KUKA KRL program: MyProgram_092().src

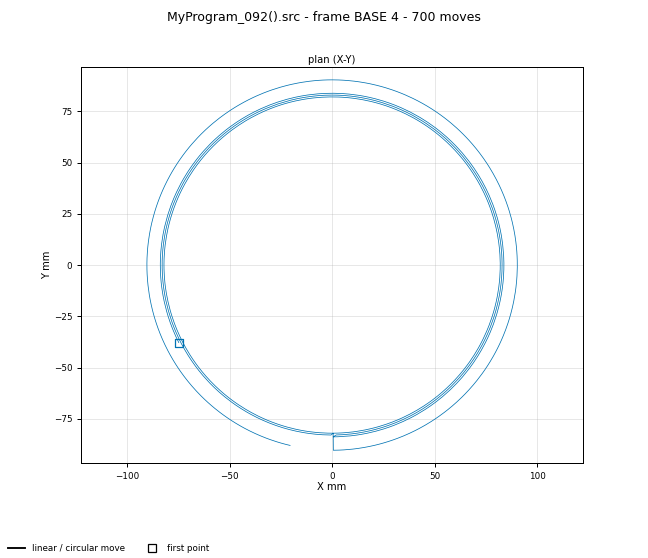
[picture p0: tool path of MyProgram_092().src in frame BASE 4, 700 of 700 moves have a stored position in this frame; points joined in program order, loops and branches not executed]
&ACCESS RVP
&REL 1
&PARAM TEMPLATE = C:\KRC\Roboter\Template\vorgabe
&PARAM EDITMASK = *
DEF MyProgram_092()
; ---- Setting reference (Base) ----
$BASE = BASE_DATA[4]

; --------------------------
; ---- Setting tool (TCP) ----
$TOOL = TOOL_DATA[3]
; --------------------------

$VEL.CP = VEL_APROX_PRINT
Startdeposition()
$VEL.CP = VEL_PRINT
LIN {X -74.828,Y -37.8282,Z 87,A -158.7584,B 24.9189,C -2.0802,E1 24.8563,E2 243.6594} C_DIS
LIN {X -76.2325,Y -34.9131,Z 87,A -161.0575,B 24.9186,C -2.084,E1 24.8536,E2 245.962} C_DIS
LIN {X -77.7703,Y -31.3357,Z 87,A -163.8809,B 24.9183,C -2.0873,E1 24.8506,E2 248.7932} C_DIS
LIN {X -78.9715,Y -28.1737,Z 87,A -166.4538,B 24.9183,C -2.0871,E1 24.8481,E2 251.3812} C_DIS
LIN {X -80.015,Y -25.0533,Z 87,A -168.1806,B 24.9167,C -2.1077,E1 24.8467,E2 253.0687} C_DIS
LIN {X -80.7299,Y -22.6451,Z 87,A -169.9657,B 24.9164,C -2.111,E1 24.8453,E2 254.8562} C_DIS
LIN {X -81.9682,Y -17.6447,Z 87,A -173.2787,B 24.9151,C -2.1273,E1 24.8432,E2 258.1497} C_DIS
LIN {X -82.5461,Y -14.7049,Z 87,A -175.5042,B 24.9151,C -2.1289,E1 24.842,E2 260.3846} C_DIS
LIN {X -83.1122,Y -11.0688,Z 87,A -177.8414,B 24.914,C -2.1414,E1 24.8411,E2 262.7057} C_DIS
LIN {X -83.3919,Y -8.7092,Z 87,A -179.5472,B 24.9138,C -2.1444,E1 24.8405,E2 264.4148} C_DIS
LIN {X -83.6299,Y -6.0204,Z 87,A 178.4494,B 24.9136,C -2.146,E1 24.8401,E2 266.4264} C_DIS
LIN {X -83.7977,Y -2.8427,Z 87,A 176.1823,B 24.9133,C -2.1504,E1 24.8398,E2 268.6965} C_DIS
LIN {X -83.8443,Y 0.5678,Z 87,A 174.0248,B 24.9123,C -2.1624,E1 24.8398,E2 270.8383} C_DIS
LIN {X -83.7774,Y 3.3843,Z 87,A 172.0675,B 24.9119,C -2.1678,E1 24.84,E2 272.7947} C_DIS
LIN {X -83.5899,Y 6.5428,Z 87,A 169.334,B 24.9125,C -2.1596,E1 24.8405,E2 275.5641} C_DIS
LIN {X -83.2161,Y 10.2664,Z 87,A 166.7868,B 24.9118,C -2.168,E1 24.8414,E2 278.1066} C_DIS
LIN {X -82.5012,Y 14.9543,Z 87,A 163.3356,B 24.9114,C -2.1728,E1 24.843,E2 281.5668} C_DIS
LIN {X -81.7692,Y 18.5465,Z 87,A 161.7678,B 24.9088,C -2.2054,E1 24.8439,E2 283.0659} C_DIS
LIN {X -80.2055,Y 24.4398,Z 87,A 157.3428,B 24.9083,C -2.2116,E1 24.8472,E2 287.5019} C_DIS
LIN {X -78.6612,Y 29.0272,Z 87,A 154.246,B 24.9069,C -2.2274,E1 24.8499,E2 290.5785} C_DIS
LIN {X -77.2818,Y 32.5206,Z 87,A 151.4219,B 24.9069,C -2.2283,E1 24.8529,E2 293.4163} C_DIS
LIN {X -75.9355,Y 35.5514,Z 87,A 148.0998,B 24.9086,C -2.2072,E1 24.8569,E2 296.8069} C_DIS
LIN {X -73.8493,Y 39.7045,Z 87,A 146.1931,B 24.905,C -2.2501,E1 24.8592,E2 298.6214} C_DIS
LIN {X -72.4886,Y 42.1385,Z 87,A 144.1984,B 24.9048,C -2.2531,E1 24.862,E2 300.6192} C_DIS
LIN {X -70.5351,Y 45.3307,Z 87,A 141.4848,B 24.9045,C -2.2562,E1 24.866,E2 303.3394} C_DIS
LIN {X -68.5387,Y 48.2985,Z 87,A 138.87,B 24.9043,C -2.2583,E1 24.8701,E2 305.9622} C_DIS
LIN {X -66.2293,Y 51.4182,Z 87,A 136.4276,B 24.9032,C -2.271,E1 24.8742,E2 308.3859} C_DIS
LIN {X -64.7484,Y 53.2718,Z 87,A 134.6169,B 24.9033,C -2.2701,E1 24.8774,E2 310.2071} C_DIS
LIN {X -62.7537,Y 55.6077,Z 87,A 132.2198,B 24.9036,C -2.2674,E1 24.8818,E2 312.6217} C_DIS
LIN {X -59.4872,Y 59.088,Z 87,A 129.4081,B 24.9018,C -2.2875,E1 24.8872,E2 315.3974} C_DIS
LIN {X -57.6192,Y 60.911,Z 87,A 127.4312,B 24.9019,C -2.2865,E1 24.8912,E2 317.385} C_DIS
LIN {X -55.0222,Y 63.2665,Z 87,A 124.7933,B 24.902,C -2.2853,E1 24.8967,E2 320.0362} C_DIS
LIN {X -51.7994,Y 65.9314,Z 87,A 122.4481,B 24.9003,C -2.3055,E1 24.9017,E2 322.342} C_DIS
LIN {X -49.9627,Y 67.3352,Z 87,A 120.4367,B 24.901,C -2.2969,E1 24.9063,E2 324.3812} C_DIS
LIN {X -46.6431,Y 69.6755,Z 87,A 117.8495,B 24.9001,C -2.3076,E1 24.9122,E2 326.9517} C_DIS
LIN {X -43.9616,Y 71.3981,Z 87,A 115.5051,B 24.9001,C -2.307,E1 24.9178,E2 329.3048} C_DIS
LIN {X -40.9981,Y 73.1385,Z 87,A 112.6787,B 24.9009,C -2.2979,E1 24.9247,E2 332.1612} C_DIS
LIN {X -38.0284,Y 74.7257,Z 87,A 111.0801,B 24.8989,C -2.3212,E1 24.9285,E2 333.7087} C_DIS
LIN {X -34.9535,Y 76.2138,Z 87,A 108.7935,B 24.8985,C -2.3261,E1 24.9343,E2 335.9894} C_DIS
LIN {X -30.3308,Y 78.1669,Z 87,A 104.6708,B 24.8998,C -2.3114,E1 24.945,E2 340.1564} C_DIS
LIN {X -26.6364,Y 79.5022,Z 87,A 101.4349,B 24.9008,C -2.2992,E1 24.9537,E2 343.4274} C_DIS
LIN {X -22.04,Y 80.8971,Z 87,A 99.0674,B 24.8983,C -2.3285,E1 24.9599,E2 345.729} C_DIS
LIN {X -18.0377,Y 81.8825,Z 87,A 96.3469,B 24.8978,C -2.3338,E1 24.9673,E2 348.4404} C_DIS
LIN {X -15.0523,Y 82.4836,Z 87,A 94.3269,B 24.8975,C -2.3372,E1 24.9728,E2 350.4545} C_DIS
LIN {X -11.9026,Y 82.9964,Z 87,A 91.9253,B 24.8979,C -2.3323,E1 24.9794,E2 352.8699} C_DIS
LIN {X -7.092,Y 83.546,Z 87,A 89.013,B 24.8968,C -2.3456,E1 24.9875,E2 355.7524} C_DIS
LIN {X -3.5283,Y 83.7712,Z 87,A 86.3333,B 24.8973,C -2.3395,E1 24.995,E2 358.4473} C_DIS
LIN {X 0.6383,Y 83.8431,Z 87,A 82.993,B 24.8985,C -2.3256,E1 25.0044,E2 361.8205} C_DIS
LIN {X 4.9069,Y 83.7022,Z 87,A 80.4957,B 24.8974,C -2.3382,E1 25.0113,E2 364.2872} C_DIS
LIN {X 8.2541,Y 83.4395,Z 87,A 77.7923,B 24.8985,C -2.3258,E1 25.0189,E2 367.0184} C_DIS
LIN {X 13.1274,Y 82.8121,Z 87,A 74.8322,B 24.8975,C -2.3368,E1 25.027,E2 369.9498} C_DIS
LIN {X 15.5161,Y 82.398,Z 87,A 73.2663,B 24.8974,C -2.3389,E1 25.0312,E2 371.509} C_DIS
LIN {X 18.3808,Y 81.8075,Z 87,A 71.2516,B 24.8974,C -2.3374,E1 25.0367,E2 373.5245} C_DIS
LIN {X 21.1726,Y 81.1288,Z 87,A 68.9963,B 24.8984,C -2.3274,E1 25.0429,E2 375.8001} C_DIS
LIN {X 24.9022,Y 80.0622,Z 87,A 66.3151,B 24.8986,C -2.3246,E1 25.0501,E2 378.4834} C_DIS
LIN {X 28.008,Y 79.0296,Z 87,A 64.3946,B 24.8979,C -2.3323,E1 25.0551,E2 380.3818} C_DIS
LIN {X 30.6424,Y 78.0456,Z 87,A 62.5561,B 24.8979,C -2.333,E1 25.0599,E2 382.2146} C_DIS
LIN {X 33.5893,Y 76.8234,Z 87,A 60.3428,B 24.8982,C -2.3296,E1 25.0656,E2 384.4305} C_DIS
LIN {X 37.9144,Y 74.784,Z 87,A 57.3959,B 24.8976,C -2.3357,E1 25.0729,E2 387.3554} C_DIS
LIN {X 42.9467,Y 72.0122,Z 87,A 52.651,B 24.9003,C -2.3047,E1 25.0846,E2 392.1597} C_DIS
LIN {X 46.689,Y 69.6444,Z 87,A 49.1059,B 24.9022,C -2.2837,E1 25.0929,E2 395.7426} C_DIS
LIN {X 50.6024,Y 66.8547,Z 87,A 47.0392,B 24.8993,C -2.3162,E1 25.0974,E2 397.7252} C_DIS
LIN {X 52.6102,Y 65.2862,Z 87,A 45.1077,B 24.9001,C -2.3069,E1 25.1016,E2 399.6713} C_DIS
LIN {X 55.6902,Y 62.6799,Z 87,A 42.3443,B 24.9006,C -2.3014,E1 25.1075,E2 402.437} C_DIS
LIN {X 58.1521,Y 60.402,Z 87,A 40.1346,B 24.9008,C -2.2994,E1 25.112,E2 404.6424} C_DIS
LIN {X 60.4415,Y 58.1111,Z 87,A 37.9335,B 24.9012,C -2.295,E1 25.1163,E2 406.8444} C_DIS
LIN {X 63.4897,Y 54.7666,Z 87,A 34.9971,B 24.9013,C -2.2931,E1 25.1217,E2 409.7722} C_DIS
LIN {X 66.8785,Y 50.5707,Z 87,A 30.8014,B 24.9035,C -2.2679,E1 25.1291,E2 414.0078} C_DIS
LIN {X 69.2571,Y 47.2612,Z 87,A 27.9992,B 24.9042,C -2.2603,E1 25.1335,E2 416.8142} C_DIS
LIN {X 71.484,Y 43.8202,Z 87,A 25.6091,B 24.9036,C -2.2664,E1 25.1371,E2 419.1779} C_DIS
LIN {X 73.1323,Y 41.0092,Z 87,A 22.6384,B 24.9062,C -2.2363,E1 25.1412,E2 422.2042} C_DIS
LIN {X 74.9856,Y 37.5142,Z 87,A 21.0042,B 24.9039,C -2.2637,E1 25.1432,E2 423.765} C_DIS
LIN {X 76.5866,Y 34.1275,Z 87,A 17.8198,B 24.9062,C -2.236,E1 25.147,E2 426.9976} C_DIS
LIN {X 78.3944,Y 29.7386,Z 87,A 15.0097,B 24.9058,C -2.2409,E1 25.1499,E2 429.7806} C_DIS
LIN {X 79.4552,Y 26.7757,Z 87,A 12.8323,B 24.9064,C -2.2337,E1 25.1519,E2 431.9629} C_DIS
LIN {X 80.6296,Y 22.9991,Z 87,A 10.4964,B 24.9061,C -2.2377,E1 25.1538,E2 434.2758} C_DIS
LIN {X 81.3509,Y 20.3052,Z 87,A 8.2265,B 24.9076,C -2.2198,E1 25.1554,E2 436.575} C_DIS
LIN {X 81.9523,Y 17.7173,Z 87,A 6.236,B 24.9085,C -2.2085,E1 25.1566,E2 438.5807} C_DIS
LIN {X 82.5669,Y 14.5892,Z 87,A 3.4341,B 24.9108,C -2.1812,E1 25.158,E2 441.4306} C_DIS
LIN {X 83.189,Y 10.4759,Z 87,A 1.7178,B 24.9084,C -2.2095,E1 25.1586,E2 443.07} C_DIS
LIN {X 83.7136,Y 4.7009,Z 87,A -2.934,B 24.9113,C -2.174,E1 25.1597,E2 447.7778} C_DIS
LIN {X 83.8404,Y 1.0489,Z 87,A -5.0144,B 24.9109,C -2.1799,E1 25.1597,E2 449.8321} C_DIS
LIN {X 83.8191,Y -2.1448,Z 87,A -7.5399,B 24.9124,C -2.1615,E1 25.1597,E2 452.3859} C_DIS
LIN {X 83.5794,Y -6.6751,Z 87,A -9.8264,B 24.911,C -2.1787,E1 25.1593,E2 454.6182} C_DIS
LIN {X 83.4163,Y -8.4761,Z 87,A -11.4575,B 24.9124,C -2.1615,E1 25.1588,E2 456.2802} C_DIS
LIN {X 83.0474,Y -11.544,Z 87,A -13.6156,B 24.913,C -2.1532,E1 25.158,E2 458.4452} C_DIS
LIN {X 82.5791,Y -14.5209,Z 87,A -15.9008,B 24.9142,C -2.1391,E1 25.157,E2 460.7502} C_DIS
LIN {X 81.9838,Y -17.5729,Z 87,A -17.866,B 24.9142,C -2.1377,E1 25.1558,E2 462.7074} C_DIS
LIN {X 81.313,Y -20.4558,Z 87,A -19.812,B 24.9146,C -2.1338,E1 25.1546,E2 464.6513} C_DIS
LIN {X 80.3605,Y -23.9219,Z 87,A -22.3448,B 24.9154,C -2.1236,E1 25.1526,E2 467.1937} C_DIS
LIN {X 78.7126,Y -28.8862,Z 87,A -25.921,B 24.9163,C -2.1125,E1 25.1493,E2 470.776} C_DIS
LIN {X 77.1528,Y -32.8265,Z 87,A -28.5213,B 24.9163,C -2.1135,E1 25.1466,E2 473.3596} C_DIS
LIN {X 75.9875,Y -35.4396,Z 87,A -30.4331,B 24.9166,C -2.1091,E1 25.1444,E2 475.2714} C_DIS
LIN {X 74.7718,Y -37.9382,Z 87,A -32.4306,B 24.9173,C -2.1002,E1 25.1419,E2 477.2793} C_DIS
LIN {X 72.8887,Y -41.4421,Z 87,A -35.7705,B 24.9195,C -2.0718,E1 25.1373,E2 480.6688} C_DIS
LIN {X 71.0423,Y -44.5317,Z 87,A -36.981,B 24.9168,C -2.1061,E1 25.1357,E2 481.7921} C_DIS
LIN {X 69.0379,Y -47.581,Z 87,A -40.7724,B 24.9207,C -2.0564,E1 25.1296,E2 485.6823} C_DIS
LIN {X 66.7405,Y -50.7544,Z 87,A -42.5288,B 24.9189,C -2.0793,E1 25.1268,E2 487.3761} C_DIS
LIN {X 63.5469,Y -54.6995,Z 87,A -45.9705,B 24.9196,C -2.0711,E1 25.1207,E2 490.8213} C_DIS
LIN {X 60.8605,Y -57.6712,Z 87,A -49.0996,B 24.9211,C -2.0514,E1 25.1147,E2 493.9831} C_DIS
LIN {X 57.5073,Y -61.0159,Z 87,A -52.4737,B 24.922,C -2.0392,E1 25.1079,E2 497.3719} C_DIS
LIN {X 53.8408,Y -64.2749,Z 87,A -55.8308,B 24.9226,C -2.0315,E1 25.1008,E2 500.7341} C_DIS
LIN {X 50.8148,Y -66.6943,Z 87,A -58.1456,B 24.9222,C -2.0365,E1 25.0957,E2 503.0285} C_DIS
LIN {X 48.0518,Y -68.7106,Z 87,A -60.3818,B 24.9223,C -2.035,E1 25.0906,E2 505.2604} C_DIS
LIN {X 45.4502,Y -70.4584,Z 87,A -62.9978,B 24.9238,C -2.0157,E1 25.0844,E2 507.9135} C_DIS
LIN {X 41.4241,Y -72.899,Z 87,A -65.5057,B 24.9225,C -2.0325,E1 25.0785,E2 510.374} C_DIS
LIN {X 38.4643,Y -74.5029,Z 87,A -68.3865,B 24.9242,C -2.0101,E1 25.0713,E2 513.2997} C_DIS
LIN {X 34.5771,Y -76.3839,Z 87,A -71.066,B 24.9239,C -2.0141,E1 25.0646,E2 515.9629} C_DIS
LIN {X 30.4393,Y -78.1253,Z 87,A -73.6463,B 24.9231,C -2.0252,E1 25.058,E2 518.5111} C_DIS
LIN {X 27.8165,Y -79.0968,Z 87,A -75.7905,B 24.9238,C -2.0153,E1 25.0523,E2 520.6742} C_DIS
LIN {X 25.1905,Y -79.9728,Z 87,A -77.915,B 24.9246,C -2.0057,E1 25.0466,E2 522.8174} C_DIS
LIN {X 21.398,Y -81.0705,Z 87,A -80.6494,B 24.9249,C -2.0016,E1 25.0392,E2 525.5569} C_DIS
LIN {X 17.2616,Y -82.0504,Z 87,A -83.1614,B 24.9242,C -2.0112,E1 25.0325,E2 528.0429} C_DIS
LIN {X 13.9856,Y -82.671,Z 87,A -85.2787,B 24.9239,C -2.0143,E1 25.0267,E2 530.1503} C_DIS
LIN {X 11.7571,Y -83.0171,Z 87,A -87.2668,B 24.925,C -1.9994,E1 25.0211,E2 532.1719} C_DIS
LIN {X 8.8073,Y -83.3817,Z 87,A -89.4978,B 24.9256,C -1.9921,E1 25.0149,E2 534.4188} C_DIS
LIN {X 2.6865,Y -83.8025,Z 87,A -93.3353,B 24.9249,C -2.0012,E1 25.0042,E2 538.2331} C_DIS
LIN {X 0.5343,Y -83.8393,Z 87,A -94.3979,B 24.924,C -2.0133,E1 25.0014,E2 539.2667} C_DIS
Enddeposition()
LIN {X 0.5343,Y -83.8393,Z 87,A -94.3979,B 24.924,C -2.0133,E1 25.0014,E2 539.2667} C_DIS
Startdeposition()
$VEL.CP = VEL_PRINT
LIN {X 2.0303,Y -82.9282,Z 87,A -92.7545,B 24.9214,C -2.0477,E1 25.0062,E2 537.5421} C_DIS
LIN {X 5.2197,Y -82.788,Z 87,A -90.5523,B 24.9214,C -2.0486,E1 25.0123,E2 535.3387} C_DIS
LIN {X 9.2115,Y -82.4396,Z 87,A -87.8793,B 24.9214,C -2.0471,E1 25.0197,E2 532.6707} C_DIS
LIN {X 12.4027,Y -82.0195,Z 87,A -85.7099,B 24.9214,C -2.047,E1 25.0257,E2 530.5037} C_DIS
LIN {X 15.4627,Y -81.4979,Z 87,A -83.588,B 24.9214,C -2.048,E1 25.0315,E2 528.3817} C_DIS
LIN {X 18.716,Y -80.8125,Z 87,A -81.2561,B 24.9211,C -2.0512,E1 25.0379,E2 526.0453} C_DIS
LIN {X 21.1632,Y -80.2079,Z 87,A -79.4671,B 24.9209,C -2.0545,E1 25.0428,E2 524.2513} C_DIS
LIN {X 24.3745,Y -79.2898,Z 87,A -77.2416,B 24.9209,C -2.0545,E1 25.0487,E2 522.0296} C_DIS
LIN {X 27.1885,Y -78.3698,Z 87,A -74.9518,B 24.92,C -2.0648,E1 25.0548,E2 519.7197} C_DIS
LIN {X 31.0208,Y -76.9333,Z 87,A -71.7524,B 24.9188,C -2.0807,E1 25.0632,E2 516.49} C_DIS
LIN {X 34.246,Y -75.5526,Z 87,A -69.5188,B 24.919,C -2.0783,E1 25.0689,E2 514.2677} C_DIS
LIN {X 38.1341,Y -73.6677,Z 87,A -66.9202,B 24.9196,C -2.0707,E1 25.0753,E2 511.694} C_DIS
LIN {X 41.09,Y -72.06,Z 87,A -64.6583,B 24.9194,C -2.0728,E1 25.0808,E2 509.4339} C_DIS
LIN {X 43.8418,Y -70.4192,Z 87,A -62.5391,B 24.9194,C -2.0739,E1 25.0858,E2 507.3186} C_DIS
LIN {X 46.18,Y -68.9094,Z 87,A -60.573,B 24.9189,C -2.079,E1 25.0904,E2 505.3469} C_DIS
LIN {X 48.4601,Y -67.3253,Z 87,A -58.5902,B 24.9185,C -2.0851,E1 25.095,E2 503.3568} C_DIS
LIN {X 51.0324,Y -65.398,Z 87,A -56.4095,B 24.9182,C -2.0885,E1 25.0998,E2 501.176} C_DIS
LIN {X 54.2794,Y -62.7283,Z 87,A -53.5166,B 24.9177,C -2.0946,E1 25.106,E2 498.2797} C_DIS
LIN {X 56.673,Y -60.5736,Z 87,A -51.5785,B 24.918,C -2.0904,E1 25.11,E2 496.3593} C_DIS
LIN {X 58.2405,Y -59.0677,Z 87,A -49.6757,B 24.9167,C -2.1072,E1 25.1138,E2 494.4248} C_DIS
LIN {X 62.023,Y -55.0836,Z 87,A -46.0174,B 24.9163,C -2.1121,E1 25.1208,E2 490.771} C_DIS
LIN {X 64.1643,Y -52.5746,Z 87,A -43.7644,B 24.9159,C -2.1172,E1 25.1248,E2 488.5162} C_DIS
LIN {X 66.9138,Y -49.0254,Z 87,A -40.5785,B 24.915,C -2.1284,E1 25.1302,E2 485.3193} C_DIS
LIN {X 68.8761,Y -46.2293,Z 87,A -38.408,B 24.915,C -2.1286,E1 25.1336,E2 483.1589} C_DIS
LIN {X 70.4082,Y -43.8595,Z 87,A -36.5463,B 24.9148,C -2.1312,E1 25.1364,E2 481.3004} C_DIS
LIN {X 71.4462,Y -42.1472,Z 87,A -34.9578,B 24.9139,C -2.142,E1 25.1387,E2 479.6945} C_DIS
LIN {X 73.2495,Y -38.9301,Z 87,A -32.8081,B 24.9144,C -2.1362,E1 25.1415,E2 477.5699} C_DIS
LIN {X 74.4196,Y -36.6433,Z 87,A -30.7236,B 24.9132,C -2.1517,E1 25.1442,E2 475.4597} C_DIS
LIN {X 75.8461,Y -33.594,Z 87,A -27.9877,B 24.9115,C -2.1725,E1 25.1473,E2 472.6896} C_DIS
LIN {X 77.1816,Y -30.3966,Z 87,A -24.8818,B 24.9089,C -2.2039,E1 25.1506,E2 469.5267} C_DIS
LIN {X 78.9703,Y -25.3902,Z 87,A -22.3572,B 24.9111,C -2.1765,E1 25.1527,E2 467.0812} C_DIS
LIN {X 79.9648,Y -22.063,Z 87,A -19.9789,B 24.9106,C -2.1833,E1 25.1545,E2 464.7005} C_DIS
LIN {X 80.7968,Y -18.7841,Z 87,A -17.6511,B 24.91,C -2.1904,E1 25.156,E2 462.3694} C_DIS
LIN {X 81.5397,Y -15.2453,Z 87,A -15.4226,B 24.91,C -2.1893,E1 25.1573,E2 460.1565} C_DIS
LIN {X 81.9895,Y -12.597,Z 87,A -13.4092,B 24.9092,C -2.2005,E1 25.1582,E2 458.1285} C_DIS
LIN {X 82.4219,Y -9.3631,Z 87,A -11.1424,B 24.9085,C -2.2082,E1 25.1589,E2 455.8569} C_DIS
LIN {X 82.7232,Y -6.1644,Z 87,A -8.8871,B 24.9078,C -2.2165,E1 25.1595,E2 453.5954} C_DIS
LIN {X 82.8968,Y -3.0547,Z 87,A -6.649,B 24.907,C -2.2263,E1 25.1597,E2 451.3475} C_DIS
LIN {X 82.9513,Y 0.435,Z 87,A -4.4772,B 24.907,C -2.226,E1 25.1597,E2 449.1893} C_DIS
LIN {X 82.8917,Y 3.1738,Z 87,A -2.8087,B 24.9072,C -2.2245,E1 25.1597,E2 447.5342} C_DIS
LIN {X 82.7777,Y 5.3713,Z 87,A -1.0247,B 24.906,C -2.2382,E1 25.1593,E2 445.7285} C_DIS
LIN {X 82.4587,Y 9.0379,Z 87,A 1.4067,B 24.9057,C -2.2425,E1 25.1587,E2 443.3013} C_DIS
LIN {X 82.0498,Y 12.207,Z 87,A 3.899,B 24.9043,C -2.2589,E1 25.1577,E2 440.7848} C_DIS
LIN {X 81.4309,Y 15.8105,Z 87,A 6.0369,B 24.9047,C -2.2539,E1 25.1566,E2 438.6715} C_DIS
LIN {X 80.8725,Y 18.4563,Z 87,A 8.0483,B 24.9038,C -2.2644,E1 25.1554,E2 436.6469} C_DIS
LIN {X 80.0446,Y 21.7676,Z 87,A 10.4184,B 24.9032,C -2.272,E1 25.1538,E2 434.2726} C_DIS
LIN {X 79.0553,Y 25.1275,Z 87,A 12.775,B 24.9027,C -2.2771,E1 25.1518,E2 431.9172} C_DIS
LIN {X 78.0708,Y 28.0369,Z 87,A 14.9855,B 24.9019,C -2.2863,E1 25.1498,E2 429.6975} C_DIS
LIN {X 76.054,Y 33.117,Z 87,A 18.5794,B 24.9015,C -2.2912,E1 25.146,E2 426.112} C_DIS
LIN {X 74.7884,Y 35.8838,Z 87,A 20.6652,B 24.901,C -2.2965,E1 25.1435,E2 424.0247} C_DIS
LIN {X 73.4664,Y 38.5184,Z 87,A 23.0021,B 24.8997,C -2.312,E1 25.1405,E2 421.6636} C_DIS
LIN {X 71.5716,Y 41.9351,Z 87,A 25.4554,B 24.8997,C -2.3112,E1 25.1371,E2 419.225} C_DIS
LIN {X 69.8041,Y 44.8145,Z 87,A 28.0717,B 24.8984,C -2.3265,E1 25.1332,E2 416.5857} C_DIS
LIN {X 67.3322,Y 48.4503,Z 87,A 30.597,B 24.8992,C -2.3174,E1 25.1292,E2 414.0943} C_DIS
LIN {X 64.0409,Y 52.7244,Z 87,A 34.4979,B 24.898,C -2.3319,E1 25.1225,E2 410.1774} C_DIS
LIN {X 61.9254,Y 55.1927,Z 87,A 36.7043,B 24.8976,C -2.3357,E1 25.1184,E2 407.9718} C_DIS
LIN {X 59.7078,Y 57.5841,Z 87,A 38.9582,B 24.8972,C -2.3407,E1 25.1141,E2 405.716} C_DIS
LIN {X 57.3682,Y 59.9159,Z 87,A 41.2709,B 24.8967,C -2.3464,E1 25.1095,E2 403.3994} C_DIS
LIN {X 54.9522,Y 62.1406,Z 87,A 43.5531,B 24.8963,C -2.3514,E1 25.1047,E2 401.1148} C_DIS
LIN {X 52.348,Y 64.348,Z 87,A 45.8038,B 24.8962,C -2.3524,E1 25.0999,E2 398.8702} C_DIS
LIN {X 50.1388,Y 66.0849,Z 87,A 48.2479,B 24.8944,C -2.3719,E1 25.0944,E2 396.3888} C_DIS
LIN {X 46.0808,Y 68.9765,Z 87,A 51.2523,B 24.8952,C -2.3637,E1 25.0876,E2 393.4143} C_DIS
LIN {X 43.7314,Y 70.4882,Z 87,A 54.2926,B 24.8917,C -2.4019,E1 25.0802,E2 390.2929} C_DIS
LIN {X 39.2055,Y 73.1029,Z 87,A 56.8142,B 24.8944,C -2.3723,E1 25.0742,E2 387.8489} C_DIS
LIN {X 36.9505,Y 74.2673,Z 87,A 58.4446,B 24.8945,C -2.3707,E1 25.0701,E2 386.2267} C_DIS
LIN {X 34.1298,Y 75.605,Z 87,A 60.5687,B 24.8945,C -2.3722,E1 25.0647,E2 384.1045} C_DIS
LIN {X 31.2785,Y 76.8284,Z 87,A 62.7084,B 24.8942,C -2.3743,E1 25.0592,E2 381.9646} C_DIS
LIN {X 29.1634,Y 77.6563,Z 87,A 64.4326,B 24.8937,C -2.3806,E1 25.0547,E2 380.2293} C_DIS
LIN {X 24.3553,Y 79.2958,Z 87,A 67.8703,B 24.8936,C -2.3812,E1 25.0456,E2 376.7966} C_DIS
LIN {X 21.0425,Y 80.2392,Z 87,A 70.1297,B 24.8938,C -2.3791,E1 25.0395,E2 374.5459} C_DIS
LIN {X 18.1801,Y 80.9363,Z 87,A 72.3313,B 24.8932,C -2.3853,E1 25.0335,E2 372.3328} C_DIS
LIN {X 14.7392,Y 81.6316,Z 87,A 74.6646,B 24.8934,C -2.3835,E1 25.0271,E2 370.0063} C_DIS
LIN {X 11.4815,Y 82.1533,Z 87,A 76.7094,B 24.894,C -2.3771,E1 25.0215,E2 367.9787} C_DIS
LIN {X 8.9508,Y 82.4678,Z 87,A 78.7829,B 24.8931,C -2.3868,E1 25.0157,E2 365.8837} C_DIS
LIN {X 5.6208,Y 82.7609,Z 87,A 80.9316,B 24.8935,C -2.3821,E1 25.0098,E2 363.7472} C_DIS
LIN {X 2.7865,Y 82.905,Z 87,A 82.9017,B 24.8935,C -2.3823,E1 25.0043,E2 361.7772} C_DIS
LIN {X -0.1777,Y 82.952,Z 87,A 85.1455,B 24.893,C -2.3877,E1 24.998,E2 359.5207} C_DIS
LIN {X -3.7837,Y 82.8655,Z 87,A 87.4949,B 24.8935,C -2.3828,E1 24.9914,E2 357.1827} C_DIS
LIN {X -6.8228,Y 82.6707,Z 87,A 89.6702,B 24.8933,C -2.384,E1 24.9854,E2 355.0036} C_DIS
LIN {X -10.4393,Y 82.2923,Z 87,A 92.1585,B 24.8935,C -2.3819,E1 24.9785,E2 352.5186} C_DIS
LIN {X -13.8683,Y 81.7842,Z 87,A 94.5707,B 24.8936,C -2.3808,E1 24.9718,E2 350.1069} C_DIS
LIN {X -17.1662,Y 81.1568,Z 87,A 96.9107,B 24.8938,C -2.3795,E1 24.9654,E2 347.7674} C_DIS
LIN {X -20.3639,Y 80.4136,Z 87,A 99.0088,B 24.8944,C -2.3724,E1 24.9598,E2 345.6831} C_DIS
LIN {X -26.45,Y 78.6216,Z 87,A 103.2611,B 24.8952,C -2.3638,E1 24.9485,E2 341.4441} C_DIS
LIN {X -32.0356,Y 76.5161,Z 87,A 107.6454,B 24.895,C -2.3657,E1 24.937,E2 337.0461} C_DIS
LIN {X -34.9479,Y 75.2303,Z 87,A 109.7374,B 24.8955,C -2.3594,E1 24.9317,E2 334.9639} C_DIS
LIN {X -37.4616,Y 74.0114,Z 87,A 112.486,B 24.8938,C -2.3795,E1 24.9247,E2 332.1602} C_DIS
LIN {X -40.7218,Y 72.2688,Z 87,A 114.1879,B 24.8963,C -2.3511,E1 24.9207,E2 330.5211} C_DIS
LIN {X -43.0757,Y 70.8903,Z 87,A 116.1714,B 24.8963,C -2.3505,E1 24.9159,E2 328.5329} C_DIS
LIN {X -45.6981,Y 69.2288,Z 87,A 118.4233,B 24.8964,C -2.3494,E1 24.9106,E2 326.2764} C_DIS
LIN {X -47.7925,Y 67.8016,Z 87,A 120.2348,B 24.8966,C -2.3476,E1 24.9065,E2 324.4629} C_DIS
LIN {X -50.488,Y 65.8175,Z 87,A 122.481,B 24.8972,C -2.341,E1 24.9015,E2 322.2244} C_DIS
LIN {X -52.8051,Y 63.9738,Z 87,A 124.6217,B 24.8973,C -2.3392,E1 24.8968,E2 320.0799} C_DIS
LIN {X -55.4324,Y 61.7108,Z 87,A 126.9488,B 24.898,C -2.3319,E1 24.892,E2 317.7609} C_DIS
LIN {X -57.7727,Y 59.526,Z 87,A 129.1821,B 24.8984,C -2.3273,E1 24.8874,E2 315.5293} C_DIS
LIN {X -59.9644,Y 57.3179,Z 87,A 131.1846,B 24.8992,C -2.3181,E1 24.8836,E2 313.5402} C_DIS
LIN {X -61.7813,Y 55.3536,Z 87,A 133.165,B 24.8992,C -2.3172,E1 24.8798,E2 311.5534} C_DIS
LIN {X -63.8978,Y 52.8965,Z 87,A 135.5169,B 24.8995,C -2.3145,E1 24.8756,E2 309.1971} C_DIS
LIN {X -65.8963,Y 50.3858,Z 87,A 137.7965,B 24.8999,C -2.3103,E1 24.8717,E2 306.9167} C_DIS
LIN {X -68.025,Y 47.4718,Z 87,A 140.1938,B 24.9007,C -2.301,E1 24.8678,E2 304.5299} C_DIS
LIN {X -69.9349,Y 44.6107,Z 87,A 142.6244,B 24.9011,C -2.2958,E1 24.8641,E2 302.0994} C_DIS
LIN {X -71.7119,Y 41.6957,Z 87,A 145.0515,B 24.9015,C -2.291,E1 24.8606,E2 299.6713} C_DIS
LIN {X -72.9229,Y 39.5373,Z 87,A 146.8911,B 24.9017,C -2.2896,E1 24.8582,E2 297.8254} C_DIS
LIN {X -74.8403,Y 35.7758,Z 87,A 149.6285,B 24.9028,C -2.2762,E1 24.8548,E2 295.1052} C_DIS
LIN {X -76.1589,Y 32.8764,Z 87,A 151.817,B 24.9034,C -2.2692,E1 24.8523,E2 292.9212} C_DIS
LIN {X -77.3285,Y 30.0226,Z 87,A 153.9695,B 24.9039,C -2.2634,E1 24.8501,E2 290.7707} C_DIS
LIN {X -78.1328,Y 27.864,Z 87,A 155.7591,B 24.9039,C -2.2638,E1 24.8484,E2 288.97} C_DIS
LIN {X -79.2818,Y 24.4005,Z 87,A 157.9673,B 24.9052,C -2.2476,E1 24.8466,E2 286.7877} C_DIS
LIN {X -80.4302,Y 20.2995,Z 87,A 161.1195,B 24.9055,C -2.244,E1 24.8443,E2 283.6257} C_DIS
LIN {X -81.1951,Y 16.9823,Z 87,A 163.3708,B 24.9064,C -2.2339,E1 24.8429,E2 281.3853} C_DIS
LIN {X -81.6924,Y 14.4008,Z 87,A 166.1527,B 24.9047,C -2.2542,E1 24.8416,E2 278.5386} C_DIS
LIN {X -82.3351,Y 10.1044,Z 87,A 168.0719,B 24.9079,C -2.2155,E1 24.8409,E2 276.7002} C_DIS
LIN {X -82.6217,Y 7.3928,Z 87,A 170.0209,B 24.9083,C -2.2112,E1 24.8403,E2 274.7498} C_DIS
LIN {X -82.826,Y 4.5621,Z 87,A 172.1823,B 24.9083,C -2.2103,E1 24.8399,E2 272.5775} C_DIS
LIN {X -82.929,Y 1.9851,Z 87,A 173.9867,B 24.9088,C -2.2052,E1 24.8398,E2 270.7744} C_DIS
LIN {X -82.9391,Y -1.4351,Z 87,A 176.2934,B 24.9095,C -2.1962,E1 24.8398,E2 268.4753} C_DIS
LIN {X -82.818,Y -4.7053,Z 87,A 178.6319,B 24.9099,C -2.1912,E1 24.8401,E2 266.1349} C_DIS
LIN {X -82.562,Y -8.0399,Z 87,A -178.9963,B 24.9104,C -2.1855,E1 24.8407,E2 263.7624} C_DIS
LIN {X -82.1491,Y -11.5111,Z 87,A -176.5205,B 24.9109,C -2.1796,E1 24.8416,E2 261.2859} C_DIS
LIN {X -81.6086,Y -14.8669,Z 87,A -174.2082,B 24.9116,C -2.1713,E1 24.8427,E2 258.9795} C_DIS
LIN {X -81.1223,Y -17.3277,Z 87,A -171.3463,B 24.9095,C -2.1967,E1 24.8445,E2 256.0402} C_DIS
LIN {X -79.8771,Y -22.3756,Z 87,A -169.2604,B 24.9137,C -2.1449,E1 24.8459,E2 254.0658} C_DIS
LIN {X -78.0902,Y -27.9838,Z 87,A -164.8484,B 24.9139,C -2.1421,E1 24.8497,E2 249.6352} C_DIS
LIN {X -77.0802,Y -30.6549,Z 87,A -162.9153,B 24.9145,C -2.1353,E1 24.8517,E2 247.7074} C_DIS
LIN {X -76.254,Y -32.6574,Z 87,A -161.2396,B 24.9145,C -2.1359,E1 24.8535,E2 246.0211} C_DIS
LIN {X -74.8397,Y -35.7771,Z 87,A -158.9227,B 24.9151,C -2.128,E1 24.8562,E2 243.7105} C_DIS
LIN {X -73.4395,Y -38.5693,Z 87,A -157.0916,B 24.9163,C -2.1132,E1 24.8585,E2 241.9049} C_DIS
LIN {X -71.9383,Y -41.3017,Z 87,A -154.555,B 24.9159,C -2.1179,E1 24.862,E2 239.3438} C_DIS
LIN {X -70.2831,Y -44.0597,Z 87,A -152.447,B 24.9166,C -2.109,E1 24.8651,E2 237.2463} C_DIS
LIN {X -68.6805,Y -46.5181,Z 87,A -150.4112,B 24.917,C -2.1041,E1 24.8682,E2 235.212} C_DIS
LIN {X -66.8277,Y -49.1431,Z 87,A -147.9073,B 24.9168,C -2.1065,E1 24.8723,E2 232.6901} C_DIS
LIN {X -64.94,Y -51.612,Z 87,A -145.4121,B 24.9164,C -2.1111,E1 24.8767,E2 230.1721} C_DIS
LIN {X -62.8613,Y -54.1257,Z 87,A -143.1524,B 24.9168,C -2.1062,E1 24.8808,E2 227.9139} C_DIS
LIN {X -59.7573,Y -57.5328,Z 87,A -140.4547,B 24.9184,C -2.0856,E1 24.8859,E2 225.2535} C_DIS
LIN {X -57.6209,Y -59.6723,Z 87,A -138.3625,B 24.9188,C -2.0814,E1 24.8901,E2 223.1626} C_DIS
LIN {X -55.0937,Y -62.014,Z 87,A -136.1182,B 24.9194,C -2.0728,E1 24.8947,E2 220.9296} C_DIS
LIN {X -52.429,Y -64.2818,Z 87,A -132.6944,B 24.9175,C -2.0971,E1 24.9022,E2 217.4351} C_DIS
LIN {X -49.0545,Y -66.8925,Z 87,A -130.7222,B 24.9201,C -2.064,E1 24.9065,E2 215.5346} C_DIS
LIN {X -47.0348,Y -68.3288,Z 87,A -129.0269,B 24.9204,C -2.0607,E1 24.9103,E2 213.8413} C_DIS
LIN {X -44.6629,Y -69.9014,Z 87,A -126.3562,B 24.919,C -2.078,E1 24.9167,E2 211.1209} C_DIS
LIN {X -41.7895,Y -71.6577,Z 87,A -124.4852,B 24.9203,C -2.0615,E1 24.9212,E2 209.2835} C_DIS
LIN {X -39.5934,Y -72.8925,Z 87,A -122.8764,B 24.9208,C -2.0554,E1 24.9251,E2 207.6847} C_DIS
LIN {X -36.9149,Y -74.2849,Z 87,A -120.7893,B 24.921,C -2.0528,E1 24.9303,E2 205.598} C_DIS
LIN {X -34.0445,Y -75.6434,Z 87,A -118.5872,B 24.9211,C -2.0506,E1 24.9358,E2 203.3958} C_DIS
LIN {X -30.7689,Y -77.0354,Z 87,A -116.2854,B 24.9217,C -2.0435,E1 24.9418,E2 201.1055} C_DIS
LIN {X -27.2819,Y -78.337,Z 87,A -113.4299,B 24.9212,C -2.0496,E1 24.9493,E2 198.2297} C_DIS
LIN {X -23.9968,Y -79.4058,Z 87,A -111.1753,B 24.9217,C -2.044,E1 24.9553,E2 195.9846} C_DIS
LIN {X -21.133,Y -80.2159,Z 87,A -108.9703,B 24.9214,C -2.0471,E1 24.9612,E2 193.7688} C_DIS
LIN {X -17.8061,Y -81.018,Z 87,A -106.6447,B 24.9216,C -2.0448,E1 24.9676,E2 191.4455} C_DIS
LIN {X -14.5203,Y -81.6709,Z 87,A -104.6214,B 24.9223,C -2.0353,E1 24.9731,E2 189.4428} C_DIS
LIN {X -11.9964,Y -82.0801,Z 87,A -102.5008,B 24.9215,C -2.0455,E1 24.979,E2 187.2961} C_DIS
LIN {X -8.1505,Y -82.5516,Z 87,A -99.8147,B 24.9215,C -2.0455,E1 24.9865,E2 184.6084} C_DIS
LIN {X -4.6424,Y -82.8215,Z 87,A -97.3108,B 24.9214,C -2.0478,E1 24.9934,E2 182.0982} C_DIS
LIN {X -0.5737,Y -82.9495,Z 87,A -94.8031,B 24.922,C -2.0389,E1 25.0004,E2 179.6112} C_DIS
LIN {X -0.5737,Y -82.9495,Z 87,A -94.8031,B 24.922,C -2.0389,E1 25.0004,E2 179.6112} C_DIS
Enddeposition()
LIN {X 0.5284,Y -82.0558,Z 87,A -94.4833,B 24.9219,C -2.0413,E1 25.0013,E2 179.2859} C_DIS
Startdeposition()
$VEL.CP = VEL_PRINT
LIN {X -2.0524,Y -82.0332,Z 87,A -96.5848,B 24.9226,C -2.032,E1 24.9954,E2 181.4096} C_DIS
LIN {X -4.0577,Y -81.9585,Z 87,A -97.9859,B 24.9226,C -2.0318,E1 24.9915,E2 182.8113} C_DIS
LIN {X -6.0617,Y -81.8347,Z 87,A -99.3976,B 24.9226,C -2.0315,E1 24.9875,E2 184.2242} C_DIS
LIN {X -8.0479,Y -81.6634,Z 87,A -101.0128,B 24.9231,C -2.0251,E1 24.983,E2 185.8556} C_DIS
LIN {X -11.0404,Y -81.3129,Z 87,A -102.9765,B 24.9228,C -2.0295,E1 24.9776,E2 187.8101} C_DIS
LIN {X -13.0545,Y -81.0139,Z 87,A -104.3175,B 24.9226,C -2.0322,E1 24.9739,E2 189.1458} C_DIS
LIN {X -15.3695,Y -80.6054,Z 87,A -106.1391,B 24.9229,C -2.0276,E1 24.9688,E2 190.9804} C_DIS
LIN {X -17.9826,Y -80.0644,Z 87,A -107.8258,B 24.9225,C -2.0335,E1 24.9643,E2 192.6551} C_DIS
LIN {X -19.9541,Y -79.5959,Z 87,A -109.2425,B 24.9225,C -2.0342,E1 24.9604,E2 194.072} C_DIS
LIN {X -21.885,Y -79.0869,Z 87,A -110.6393,B 24.9223,C -2.035,E1 24.9567,E2 195.4692} C_DIS
LIN {X -24.2769,Y -78.3841,Z 87,A -112.5571,B 24.9226,C -2.0312,E1 24.9515,E2 197.3993} C_DIS
LIN {X -26.7169,Y -77.5878,Z 87,A -114.4223,B 24.9226,C -2.0305,E1 24.9466,E2 199.2697} C_DIS
LIN {X -29.5376,Y -76.5585,Z 87,A -116.3624,B 24.9222,C -2.0368,E1 24.9415,E2 201.1986} C_DIS
LIN {X -31.4226,Y -75.8043,Z 87,A -117.689,B 24.9219,C -2.0408,E1 24.9381,E2 202.5187} C_DIS
LIN {X -33.8004,Y -74.7728,Z 87,A -119.5908,B 24.9219,C -2.0402,E1 24.9332,E2 204.4265} C_DIS
LIN {X -36.0044,Y -73.7384,Z 87,A -121.217,B 24.9216,C -2.0442,E1 24.9291,E2 206.0473} C_DIS
LIN {X -37.8002,Y -72.8342,Z 87,A -122.6317,B 24.9216,C -2.0457,E1 24.9256,E2 207.4623} C_DIS
LIN {X -39.5702,Y -71.888,Z 87,A -124.2959,B 24.9219,C -2.0402,E1 24.9215,E2 209.1443} C_DIS
LIN {X -42.2054,Y -70.3731,Z 87,A -126.158,B 24.9212,C -2.0505,E1 24.9171,E2 210.9877} C_DIS
LIN {X -43.9262,Y -69.312,Z 87,A -127.5652,B 24.921,C -2.0527,E1 24.9137,E2 212.394} C_DIS
LIN {X -45.6088,Y -68.2166,Z 87,A -128.9722,B 24.9208,C -2.0548,E1 24.9104,E2 213.8007} C_DIS
LIN {X -47.6929,Y -66.7744,Z 87,A -130.8552,B 24.9208,C -2.0546,E1 24.9061,E2 215.6906} C_DIS
LIN {X -50.2855,Y -64.845,Z 87,A -133.1276,B 24.9206,C -2.058,E1 24.9011,E2 217.9628} C_DIS
LIN {X -52.4824,Y -63.0796,Z 87,A -135.2318,B 24.9206,C -2.058,E1 24.8965,E2 220.0752} C_DIS
LIN {X -54.7365,Y -61.1339,Z 87,A -137.2009,B 24.92,C -2.065,E1 24.8924,E2 222.0354} C_DIS
LIN {X -56.9529,Y -59.0745,Z 87,A -139.3194,B 24.9197,C -2.0691,E1 24.8881,E2 224.1527} C_DIS
LIN {X -59.4309,Y -56.5832,Z 87,A -141.917,B 24.9197,C -2.0704,E1 24.883,E2 226.7584} C_DIS
LIN {X -61.5061,Y -54.3198,Z 87,A -144.036,B 24.9192,C -2.0758,E1 24.8791,E2 228.8739} C_DIS
LIN {X -63.4464,Y -52.0406,Z 87,A -146.1801,B 24.9189,C -2.0792,E1 24.8752,E2 231.0198} C_DIS
LIN {X -65.322,Y -49.6659,Z 87,A -148.0554,B 24.918,C -2.0906,E1 24.872,E2 232.8768} C_DIS
LIN {X -66.5099,Y -48.0636,Z 87,A -149.4653,B 24.9178,C -2.0936,E1 24.8697,E2 234.2865} C_DIS
LIN {X -67.9581,Y -45.9906,Z 87,A -151.3358,B 24.9177,C -2.0952,E1 24.8667,E2 236.1624} C_DIS
LIN {X -69.3344,Y -43.891,Z 87,A -152.994,B 24.9171,C -2.1022,E1 24.8642,E2 237.8123} C_DIS
LIN {X -70.3809,Y -42.1926,Z 87,A -154.4004,B 24.9169,C -2.1055,E1 24.8622,E2 239.218} C_DIS
LIN {X -71.4001,Y -40.4439,Z 87,A -156.0453,B 24.9171,C -2.1031,E1 24.8599,E2 240.8772} C_DIS
LIN {X -72.8381,Y -37.7929,Z 87,A -158.1226,B 24.9165,C -2.1095,E1 24.8572,E2 242.9502} C_DIS
LIN {X -74.1821,Y -35.0814,Z 87,A -160.0625,B 24.9157,C -2.12,E1 24.8548,E2 244.8756} C_DIS
LIN {X -75.0257,Y -33.2389,Z 87,A -161.4767,B 24.9154,C -2.124,E1 24.8532,E2 246.288} C_DIS
LIN {X -75.8179,Y -31.3898,Z 87,A -163.1232,B 24.9156,C -2.1216,E1 24.8514,E2 247.9493} C_DIS
LIN {X -76.9181,Y -28.5884,Z 87,A -165.0601,B 24.9147,C -2.132,E1 24.8495,E2 249.8722} C_DIS
LIN {X -77.6149,Y -26.6376,Z 87,A -166.4547,B 24.9143,C -2.1377,E1 24.8482,E2 251.2614} C_DIS
LIN {X -78.2343,Y -24.7601,Z 87,A -167.865,B 24.914,C -2.141,E1 24.847,E2 252.6718} C_DIS
LIN {X -78.9809,Y -22.2591,Z 87,A -169.7655,B 24.9138,C -2.1444,E1 24.8455,E2 254.5751} C_DIS
LIN {X -79.5983,Y -19.9447,Z 87,A -171.3798,B 24.9132,C -2.151,E1 24.8444,E2 256.1831} C_DIS
LIN {X -80.0559,Y -18.0197,Z 87,A -172.772,B 24.9129,C -2.1549,E1 24.8435,E2 257.574} C_DIS
LIN {X -80.4847,Y -15.9963,Z 87,A -174.2174,B 24.9125,C -2.1593,E1 24.8427,E2 259.0174} C_DIS
LIN {X -80.8502,Y -14.0329,Z 87,A -175.8315,B 24.9127,C -2.158,E1 24.8419,E2 260.6444} C_DIS
LIN {X -81.3131,Y -11.039,Z 87,A -177.768,B 24.9117,C -2.1692,E1 24.8411,E2 262.5657} C_DIS
LIN {X -81.5608,Y -9.0281,Z 87,A -179.1734,B 24.9114,C -2.1739,E1 24.8407,E2 263.9683} C_DIS
LIN {X -81.8376,Y -6.0238,Z 87,A 178.7027,B 24.9109,C -2.1801,E1 24.8402,E2 266.09} C_DIS
LIN {X -81.9607,Y -4.0162,Z 87,A 177.2433,B 24.9106,C -2.1831,E1 24.8399,E2 267.551} C_DIS
LIN {X -82.0347,Y -1.9946,Z 87,A 175.8443,B 24.9102,C -2.188,E1 24.8399,E2 268.9469} C_DIS
LIN {X -82.0574,Y 0.413,Z 87,A 173.9804,B 24.9102,C -2.1886,E1 24.8398,E2 270.8205} C_DIS
LIN {X -82.0035,Y 3.0189,Z 87,A 172.3234,B 24.9093,C -2.1986,E1 24.8399,E2 272.4636} C_DIS
LIN {X -81.9048,Y 5.0281,Z 87,A 170.9105,B 24.909,C -2.2029,E1 24.8401,E2 273.8748} C_DIS
LIN {X -81.7557,Y 7.0489,Z 87,A 169.3818,B 24.9088,C -2.2044,E1 24.8405,E2 275.4089} C_DIS
LIN {X -81.4668,Y 9.8322,Z 87,A 167.4743,B 24.9082,C -2.2119,E1 24.8411,E2 277.31} C_DIS
LIN {X -81.1636,Y 12.088,Z 87,A 165.927,B 24.9077,C -2.218,E1 24.8417,E2 278.8519} C_DIS
LIN {X -80.8445,Y 14.0647,Z 87,A 164.528,B 24.9073,C -2.2224,E1 24.8423,E2 280.2487} C_DIS
LIN {X -80.4769,Y 16.0353,Z 87,A 163.1084,B 24.907,C -2.2264,E1 24.8431,E2 281.6674} C_DIS
LIN {X -80.0643,Y 17.9829,Z 87,A 161.7082,B 24.9067,C -2.2305,E1 24.8439,E2 283.0659} C_DIS
LIN {X -79.5972,Y 19.9489,Z 87,A 160.0332,B 24.9069,C -2.2281,E1 24.845,E2 284.7564} C_DIS
LIN {X -78.8105,Y 22.86,Z 87,A 158.1566,B 24.9058,C -2.2406,E1 24.8464,E2 286.6141} C_DIS
LIN {X -78.2229,Y 24.7962,Z 87,A 156.5932,B 24.9058,C -2.2411,E1 24.8477,E2 288.1853} C_DIS
LIN {X -77.2655,Y 27.6356,Z 87,A 154.3939,B 24.9055,C -2.2448,E1 24.8497,E2 290.3884} C_DIS
LIN {X -76.1925,Y 30.4696,Z 87,A 152.4967,B 24.9044,C -2.2569,E1 24.8516,E2 292.2673} C_DIS
LIN {X -75.2949,Y 32.6212,Z 87,A 150.6825,B 24.9044,C -2.2569,E1 24.8536,E2 294.0913} C_DIS
LIN {X -74.1846,Y 35.0761,Z 87,A 148.9655,B 24.9036,C -2.2668,E1 24.8556,E2 295.7942} C_DIS
LIN {X -73.0792,Y 37.321,Z 87,A 147.0558,B 24.9036,C -2.2677,E1 24.858,E2 297.7119} C_DIS
LIN {X -71.8777,Y 39.5887,Z 87,A 145.4209,B 24.9027,C -2.277,E1 24.8602,E2 299.3333} C_DIS
LIN {X -70.8864,Y 41.3375,Z 87,A 144.0075,B 24.9024,C -2.2808,E1 24.8621,E2 300.7451} C_DIS
LIN {X -69.8597,Y 43.0501,Z 87,A 142.5851,B 24.9021,C -2.284,E1 24.8642,E2 302.1672} C_DIS
LIN {X -68.7834,Y 44.7496,Z 87,A 141.1717,B 24.9018,C -2.2876,E1 24.8663,E2 303.579} C_DIS
LIN {X -67.6658,Y 46.4223,Z 87,A 139.5805,B 24.9019,C -2.2866,E1 24.8688,E2 305.1806} C_DIS
LIN {X -65.9051,Y 48.8896,Z 87,A 137.4206,B 24.9015,C -2.2912,E1 24.8724,E2 307.34} C_DIS
LIN {X -64.0593,Y 51.2843,Z 87,A 135.2972,B 24.9011,C -2.2964,E1 24.8761,E2 309.4609} C_DIS
LIN {X -62.1361,Y 53.5984,Z 87,A 133.1813,B 24.9006,C -2.3014,E1 24.8799,E2 311.5746} C_DIS
LIN {X -60.1131,Y 55.8578,Z 87,A 131.0531,B 24.9002,C -2.3064,E1 24.8839,E2 313.7003} C_DIS
LIN {X -58.0201,Y 58.0288,Z 87,A 128.9367,B 24.8998,C -2.3112,E1 24.888,E2 315.8143} C_DIS
LIN {X -55.843,Y 60.1268,Z 87,A 126.8148,B 24.8994,C -2.3158,E1 24.8923,E2 317.9339} C_DIS
LIN {X -53.6013,Y 62.1336,Z 87,A 124.6965,B 24.899,C -2.3201,E1 24.8968,E2 320.0505} C_DIS
LIN {X -51.2704,Y 64.0705,Z 87,A 122.5767,B 24.8986,C -2.3245,E1 24.9013,E2 322.1676} C_DIS
LIN {X -48.8686,Y 65.9206,Z 87,A 120.6784,B 24.8977,C -2.3348,E1 24.9055,E2 324.0482} C_DIS
LIN {X -47.2382,Y 67.0986,Z 87,A 119.2667,B 24.8975,C -2.3375,E1 24.9087,E2 325.4585} C_DIS
LIN {X -45.5795,Y 68.2363,Z 87,A 117.8546,B 24.8973,C -2.34,E1 24.912,E2 326.8693} C_DIS
LIN {X -43.8934,Y 69.3329,Z 87,A 116.4372,B 24.8971,C -2.3423,E1 24.9153,E2 328.2858} C_DIS
LIN {X -42.1842,Y 70.3859,Z 87,A 114.87,B 24.8972,C -2.3403,E1 24.9191,E2 329.8625} C_DIS
LIN {X -39.5449,Y 71.9018,Z 87,A 112.8623,B 24.8966,C -2.3472,E1 24.9239,E2 331.8596} C_DIS
LIN {X -37.7752,Y 72.8471,Z 87,A 111.4913,B 24.8963,C -2.3504,E1 24.9273,E2 333.2269} C_DIS
LIN {X -35.9686,Y 73.7558,Z 87,A 110.0836,B 24.8961,C -2.3527,E1 24.9308,E2 334.6327} C_DIS
LIN {X -33.7506,Y 74.7953,Z 87,A 108.2301,B 24.8963,C -2.3514,E1 24.9356,E2 336.494} C_DIS
LIN {X -31.3521,Y 75.8332,Z 87,A 106.5313,B 24.8957,C -2.3574,E1 24.9399,E2 338.1823} C_DIS
LIN {X -29.4982,Y 76.5736,Z 87,A 105.1413,B 24.8955,C -2.3594,E1 24.9435,E2 339.5706} C_DIS
LIN {X -27.0542,Y 77.4695,Z 87,A 103.2367,B 24.8955,C -2.3594,E1 24.9485,E2 341.4793} C_DIS
LIN {X -24.7938,Y 78.2237,Z 87,A 101.6362,B 24.8952,C -2.363,E1 24.9528,E2 343.0739} C_DIS
LIN {X -22.8676,Y 78.8083,Z 87,A 100.2275,B 24.8951,C -2.3645,E1 24.9565,E2 344.4815} C_DIS
LIN {X -20.4547,Y 79.4672,Z 87,A 98.3427,B 24.8953,C -2.3624,E1 24.9616,E2 346.374} C_DIS
LIN {X -17.9719,Y 80.0668,Z 87,A 96.6906,B 24.8948,C -2.3677,E1 24.9661,E2 348.0158} C_DIS
LIN {X -15.9896,Y 80.486,Z 87,A 95.2829,B 24.8947,C -2.369,E1 24.9699,E2 349.4219} C_DIS
LIN {X -14.0266,Y 80.8513,Z 87,A 93.8765,B 24.8947,C -2.3698,E1 24.9738,E2 350.828} C_DIS
LIN {X -11.4471,Y 81.2552,Z 87,A 91.9563,B 24.8947,C -2.3682,E1 24.9791,E2 352.7534} C_DIS
LIN {X -9.0185,Y 81.5618,Z 87,A 90.3495,B 24.8944,C -2.3721,E1 24.9836,E2 354.3521} C_DIS
LIN {X -7.0329,Y 81.7571,Z 87,A 88.9357,B 24.8944,C -2.3721,E1 24.9875,E2 355.7665} C_DIS
LIN {X -5.028,Y 81.9048,Z 87,A 87.5306,B 24.8944,C -2.3727,E1 24.9914,E2 357.1708} C_DIS
LIN {X -3.02,Y 82.0035,Z 87,A 86.0885,B 24.8944,C -2.3721,E1 24.9954,E2 358.6148} C_DIS
LIN {X -0.9737,Y 82.0531,Z 87,A 84.7155,B 24.8942,C -2.3741,E1 24.9993,E2 359.9831} C_DIS
LIN {X 1.02,Y 82.0526,Z 87,A 83.3039,B 24.8942,C -2.3737,E1 25.0032,E2 361.3954} C_DIS
LIN {X 3.0286,Y 82.0031,Z 87,A 81.8862,B 24.8942,C -2.3734,E1 25.0072,E2 362.8135} C_DIS
LIN {X 5.0358,Y 81.9044,Z 87,A 80.3329,B 24.8947,C -2.3691,E1 25.0115,E2 364.3765} C_DIS
LIN {X 8.0407,Y 81.6641,Z 87,A 78.1515,B 24.8949,C -2.3667,E1 25.0176,E2 366.5624} C_DIS
LIN {X 11.0459,Y 81.3122,Z 87,A 76.1695,B 24.8946,C -2.3701,E1 25.0231,E2 368.5348} C_DIS
LIN {X 13.056,Y 81.0136,Z 87,A 74.8715,B 24.8943,C -2.3732,E1 25.0266,E2 369.8241} C_DIS
LIN {X 15.0234,Y 80.6721,Z 87,A 73.4688,B 24.8943,C -2.3724,E1 25.0305,E2 371.2272} C_DIS
LIN {X 17.011,Y 80.2764,Z 87,A 72.0743,B 24.8943,C -2.3724,E1 25.0343,E2 372.62} C_DIS
LIN {X 18.9594,Y 79.8388,Z 87,A 70.6631,B 24.8945,C -2.3712,E1 25.0381,E2 374.0322} C_DIS
LIN {X 21.3163,Y 79.2405,Z 87,A 68.8213,B 24.895,C -2.3659,E1 25.0431,E2 375.8837} C_DIS
LIN {X 23.8591,Y 78.5136,Z 87,A 66.914,B 24.8953,C -2.3627,E1 25.0482,E2 377.7952} C_DIS
LIN {X 26.6997,Y 77.5939,Z 87,A 65.0387,B 24.8948,C -2.3673,E1 25.0532,E2 379.6561} C_DIS
LIN {X 28.5979,Y 76.9145,Z 87,A 63.647,B 24.8949,C -2.3665,E1 25.0568,E2 381.0467} C_DIS
LIN {X 31.0049,Y 75.9746,Z 87,A 61.7616,B 24.8953,C -2.3622,E1 25.0617,E2 382.9379} C_DIS
LIN {X 33.2658,Y 75.0137,Z 87,A 60.1353,B 24.8953,C -2.363,E1 25.0659,E2 384.5584} C_DIS
LIN {X 36.0099,Y 73.7357,Z 87,A 58.0269,B 24.8954,C -2.3607,E1 25.0712,E2 386.667} C_DIS
LIN {X 37.8074,Y 72.8305,Z 87,A 56.5986,B 24.8957,C -2.3582,E1 25.0748,E2 388.0972} C_DIS
LIN {X 39.6001,Y 71.8713,Z 87,A 55.2141,B 24.8957,C -2.3573,E1 25.0782,E2 389.4797} C_DIS
LIN {X 41.3533,Y 70.8771,Z 87,A 53.8194,B 24.8959,C -2.3557,E1 25.0815,E2 390.8741} C_DIS
LIN {X 43.1758,Y 69.7812,Z 87,A 52.4075,B 24.8959,C -2.3557,E1 25.0849,E2 392.2814} C_DIS
LIN {X 45.3286,Y 68.4017,Z 87,A 50.4997,B 24.8964,C -2.3492,E1 25.0894,E2 394.1986} C_DIS
LIN {X 47.2549,Y 67.0869,Z 87,A 48.9287,B 24.8965,C -2.3483,E1 25.093,E2 395.7664} C_DIS
LIN {X 49.0937,Y 65.7518,Z 87,A 47.2516,B 24.897,C -2.3427,E1 25.0968,E2 397.4505} C_DIS
LIN {X 51.2822,Y 64.061,Z 87,A 45.2027,B 24.8976,C -2.3356,E1 25.1013,E2 399.5088} C_DIS
LIN {X 53.6043,Y 62.131,Z 87,A 43.1056,B 24.898,C -2.3319,E1 25.1058,E2 401.6066} C_DIS
LIN {X 55.8517,Y 60.1188,Z 87,A 41.0054,B 24.8983,C -2.3279,E1 25.1101,E2 403.7078} C_DIS
LIN {X 58.0238,Y 58.0253,Z 87,A 38.9099,B 24.8987,C -2.3238,E1 25.1143,E2 405.8041} C_DIS
LIN {X 60.1224,Y 55.8479,Z 87,A 36.8084,B 24.8991,C -2.3195,E1 25.1183,E2 407.9066} C_DIS
LIN {X 62.1358,Y 53.5987,Z 87,A 34.6996,B 24.8995,C -2.3147,E1 25.1222,E2 410.0174} C_DIS
LIN {X 64.084,Y 51.2533,Z 87,A 32.6025,B 24.8998,C -2.3107,E1 25.1259,E2 412.1141} C_DIS
LIN {X 65.9258,Y 48.8616,Z 87,A 30.7267,B 24.8996,C -2.3129,E1 25.129,E2 413.9757} C_DIS
LIN {X 67.415,Y 46.7831,Z 87,A 28.8483,B 24.9003,C -2.3056,E1 25.1321,E2 415.8624} C_DIS
LIN {X 68.7859,Y 44.7458,Z 87,A 27.2245,B 24.9003,C -2.3041,E1 25.1346,E2 417.4817} C_DIS
LIN {X 69.8699,Y 43.0333,Z 87,A 25.8366,B 24.9006,C -2.3012,E1 25.1366,E2 418.8692} C_DIS
LIN {X 70.904,Y 41.3074,Z 87,A 24.2056,B 24.9016,C -2.2903,E1 25.1389,E2 420.5177} C_DIS
LIN {X 72.3743,Y 38.6734,Z 87,A 22.3372,B 24.9014,C -2.2922,E1 25.1414,E2 422.3717} C_DIS
LIN {X 73.3602,Y 36.7674,Z 87,A 20.9247,B 24.9015,C -2.2909,E1 25.1432,E2 423.7799} C_DIS
LIN {X 74.1814,Y 35.0828,Z 87,A 19.5473,B 24.902,C -2.285,E1 25.1449,E2 425.1638} C_DIS
LIN {X 75.2242,Y 32.7835,Z 87,A 17.6683,B 24.9028,C -2.2763,E1 25.147,E2 427.0532} C_DIS
LIN {X 76.2021,Y 30.4451,Z 87,A 15.9292,B 24.9031,C -2.2722,E1 25.1489,E2 428.7925} C_DIS
LIN {X 77.1987,Y 27.8191,Z 87,A 14.06,B 24.9034,C -2.2694,E1 25.1507,E2 430.6576} C_DIS
LIN {X 77.9168,Y 25.7421,Z 87,A 12.3359,B 24.9043,C -2.2587,E1 25.1522,E2 432.3973} C_DIS
LIN {X 78.8171,Y 22.8371,Z 87,A 10.4631,B 24.9041,C -2.2605,E1 25.1537,E2 434.2552} C_DIS
LIN {X 79.3495,Y 20.9126,Z 87,A 9.0593,B 24.9045,C -2.2559,E1 25.1548,E2 435.6617} C_DIS
LIN {X 79.8417,Y 18.9469,Z 87,A 7.6716,B 24.9048,C -2.2525,E1 25.1557,E2 437.0495} C_DIS
LIN {X 80.2791,Y 16.9986,Z 87,A 6.2666,B 24.9052,C -2.2479,E1 25.1565,E2 438.4573} C_DIS
LIN {X 80.6729,Y 15.019,Z 87,A 4.8694,B 24.9055,C -2.2439,E1 25.1573,E2 439.8557} C_DIS
LIN {X 81.0188,Y 13.0242,Z 87,A 3.4669,B 24.9059,C -2.2398,E1 25.1579,E2 441.2595} C_DIS
LIN {X 81.3185,Y 10.9972,Z 87,A 2.0713,B 24.9062,C -2.2365,E1 25.1585,E2 442.6547} C_DIS
LIN {X 81.6211,Y 8.4523,Z 87,A 0.0352,B 24.9073,C -2.2229,E1 25.1591,E2 444.7111} C_DIS
LIN {X 81.9054,Y 5.0179,Z 87,A -2.121,B 24.9073,C -2.2234,E1 25.1595,E2 446.8533} C_DIS
LIN {X 82.0037,Y 3.0115,Z 87,A -3.5139,B 24.9076,C -2.2192,E1 25.1597,E2 448.2477} C_DIS
LIN {X 82.0532,Y 0.9604,Z 87,A -4.9329,B 24.908,C -2.2151,E1 25.1597,E2 449.6679} C_DIS
LIN {X 82.0344,Y -2.0113,Z 87,A -6.9892,B 24.9085,C -2.2091,E1 25.1597,E2 451.7263} C_DIS
LIN {X 81.9589,Y -4.0507,Z 87,A -8.3934,B 24.9088,C -2.2052,E1 25.1595,E2 453.1313} C_DIS
LIN {X 81.835,Y -6.0576,Z 87,A -9.7972,B 24.9092,C -2.2007,E1 25.1593,E2 454.5373} C_DIS
LIN {X 81.6636,Y -8.0464,Z 87,A -11.4141,B 24.9101,C -2.1889,E1 25.1588,E2 456.1724} C_DIS
LIN {X 81.3127,Y -11.0423,Z 87,A -13.2811,B 24.9101,C -2.19,E1 25.1582,E2 458.0259} C_DIS
LIN {X 81.0153,Y -13.0461,Z 87,A -14.6769,B 24.9104,C -2.1861,E1 25.1576,E2 459.4226} C_DIS
LIN {X 80.674,Y -15.0128,Z 87,A -16.2334,B 24.9112,C -2.1763,E1 25.1568,E2 460.9931} C_DIS
LIN {X 80.0642,Y -17.9836,Z 87,A -18.3207,B 24.9116,C -2.1706,E1 25.1556,E2 463.0817} C_DIS
LIN {X 79.349,Y -20.9148,Z 87,A -20.2563,B 24.9117,C -2.1696,E1 25.1543,E2 465.0087} C_DIS
LIN {X 78.8125,Y -22.8534,Z 87,A -21.8819,B 24.9127,C -2.158,E1 25.153,E2 466.6523} C_DIS
LIN {X 77.9,Y -25.792,Z 87,A -23.7768,B 24.9125,C -2.1595,E1 25.1514,E2 468.5328} C_DIS
LIN {X 77.2474,Y -27.6854,Z 87,A -25.1586,B 24.9128,C -2.1558,E1 25.1502,E2 469.9157} C_DIS
LIN {X 76.5573,Y -29.5408,Z 87,A -26.7386,B 24.9137,C -2.1451,E1 25.1486,E2 471.5121} C_DIS
LIN {X 75.4187,Y -32.3372,Z 87,A -28.65,B 24.9137,C -2.1451,E1 25.1465,E2 473.413} C_DIS
LIN {X 74.5973,Y -34.1894,Z 87,A -30.0365,B 24.914,C -2.1417,E1 25.1449,E2 474.7999} C_DIS
LIN {X 73.7368,Y -36.0077,Z 87,A -31.4413,B 24.9143,C -2.1376,E1 25.1432,E2 476.207} C_DIS
LIN {X 72.8321,Y -37.8043,Z 87,A -33.0196,B 24.9151,C -2.1278,E1 25.1412,E2 477.8} C_DIS
LIN {X 71.3908,Y -40.4602,Z 87,A -34.9419,B 24.9151,C -2.1278,E1 25.1386,E2 479.7124} C_DIS
LIN {X 70.379,Y -42.1956,Z 87,A -36.4016,B 24.9156,C -2.1219,E1 25.1365,E2 481.1785} C_DIS
LIN {X 69.3168,Y -43.9187,Z 87,A -37.7215,B 24.9156,C -2.1209,E1 25.1346,E2 482.4939} C_DIS
LIN {X 68.2206,Y -45.6029,Z 87,A -39.1166,B 24.9159,C -2.1172,E1 25.1324,E2 483.8908} C_DIS
LIN {X 67.0545,Y -47.3003,Z 87,A -40.5419,B 24.9162,C -2.1137,E1 25.1302,E2 485.3174} C_DIS
LIN {X 65.8915,Y -48.9078,Z 87,A -42.1404,B 24.9171,C -2.1031,E1 25.1275,E2 486.9333} C_DIS
LIN {X 64.052,Y -51.2934,Z 87,A -44.2349,B 24.9175,C -2.0978,E1 25.1239,E2 489.0305} C_DIS
LIN {X 62.1335,Y -53.6014,Z 87,A -46.3236,B 24.9179,C -2.0926,E1 25.1201,E2 491.122} C_DIS
LIN {X 60.0908,Y -55.8814,Z 87,A -48.4392,B 24.9182,C -2.0879,E1 25.1161,E2 493.2392} C_DIS
LIN {X 58.0076,Y -58.0412,Z 87,A -50.5274,B 24.9186,C -2.083,E1 25.112,E2 495.3301} C_DIS
LIN {X 55.837,Y -60.1324,Z 87,A -52.6236,B 24.919,C -2.0783,E1 25.1078,E2 497.4288} C_DIS
LIN {X 53.6007,Y -62.1342,Z 87,A -54.7216,B 24.9194,C -2.0735,E1 25.1034,E2 499.5299} C_DIS
LIN {X 51.2624,Y -64.0768,Z 87,A -56.8214,B 24.9197,C -2.0695,E1 25.0988,E2 501.6311} C_DIS
LIN {X 48.8637,Y -65.9243,Z 87,A -58.7022,B 24.9195,C -2.0725,E1 25.0946,E2 503.4982} C_DIS
LIN {X 46.8881,Y -67.342,Z 87,A -60.5437,B 24.9201,C -2.0645,E1 25.0904,E2 505.3522} C_DIS
LIN {X 44.7514,Y -68.7823,Z 87,A -62.2012,B 24.9201,C -2.0654,E1 25.0866,E2 507.0019} C_DIS
LIN {X 43.0388,Y -69.8666,Z 87,A -63.6029,B 24.9201,C -2.0632,E1 25.0833,E2 508.4045} C_DIS
LIN {X 41.302,Y -70.907,Z 87,A -65.0116,B 24.9204,C -2.0607,E1 25.0799,E2 509.8146} C_DIS
LIN {X 39.5648,Y -71.891,Z 87,A -66.4348,B 24.9206,C -2.0574,E1 25.0764,E2 511.2415} C_DIS
LIN {X 37.7818,Y -72.8437,Z 87,A -67.9594,B 24.9211,C -2.0515,E1 25.0726,E2 512.7759} C_DIS
LIN {X 35.8152,Y -73.8295,Z 87,A -69.2942,B 24.9208,C -2.0553,E1 25.0693,E2 514.0982} C_DIS
LIN {X 34.0963,Y -74.6395,Z 87,A -70.6536,B 24.921,C -2.0522,E1 25.0658,E2 515.4614} C_DIS
LIN {X 32.2953,Y -75.4365,Z 87,A -72.2206,B 24.9216,C -2.0442,E1 25.0618,E2 517.0436} C_DIS
LIN {X 29.5251,Y -76.5634,Z 87,A -74.2988,B 24.9218,C -2.0416,E1 25.0564,E2 519.1232} C_DIS
LIN {X 26.673,Y -77.6029,Z 87,A -76.2157,B 24.9216,C -2.0451,E1 25.0514,E2 521.0279} C_DIS
LIN {X 24.7773,Y -78.2289,Z 87,A -77.7271,B 24.922,C -2.0398,E1 25.0473,E2 522.549} C_DIS
LIN {X 22.8384,Y -78.8168,Z 87,A -79.0171,B 24.9218,C -2.042,E1 25.0439,E2 523.8315} C_DIS
LIN {X 20.9141,Y -79.3492,Z 87,A -80.427,B 24.922,C -2.0401,E1 25.0401,E2 525.2438} C_DIS
LIN {X 18.7207,Y -79.8939,Z 87,A -82.178,B 24.9225,C -2.0333,E1 25.0353,E2 527.0083} C_DIS
LIN {X 15.9836,Y -80.4872,Z 87,A -83.9341,B 24.9221,C -2.0376,E1 25.0305,E2 528.752} C_DIS
LIN {X 14.0216,Y -80.8522,Z 87,A -85.3349,B 24.9222,C -2.0363,E1 25.0267,E2 530.1544} C_DIS
LIN {X 12.0218,Y -81.1736,Z 87,A -86.7373,B 24.9222,C -2.0356,E1 25.0228,E2 531.557} C_DIS
LIN {X 10.0292,Y -81.4438,Z 87,A -88.2723,B 24.9227,C -2.0308,E1 25.0185,E2 533.1022} C_DIS
LIN {X 7.0219,Y -81.758,Z 87,A -90.2661,B 24.9225,C -2.0332,E1 25.013,E2 535.0892} C_DIS
LIN {X 5.0193,Y -81.9053,Z 87,A -91.6671,B 24.9225,C -2.0326,E1 25.0091,E2 536.491} C_DIS
LIN {X 2.8654,Y -82.0082,Z 87,A -93.0776,B 24.9224,C -2.0349,E1 25.0052,E2 537.8956} C_DIS
LIN {X 0.5284,Y -82.0558,Z 87,A -94.4831,B 24.9219,C -2.0412,E1 25.0013,E2 539.2859} C_DIS
Enddeposition()
LIN {X 0.6077,Y -90.3807,Z 88,A -93.9919,B 24.931,C -1.9178,E1 25.0019,E2 539.0874} C_DIS
Startdeposition()
$VEL.CP = VEL_PRINT
LIN {X 3.5529,Y -90.3148,Z 88,A -92.0855,B 24.931,C -1.9197,E1 25.0072,E2 537.177} C_DIS
LIN {X 5.7683,Y -90.2004,Z 88,A -90.6807,B 24.9309,C -1.9202,E1 25.0111,E2 535.7714} C_DIS
LIN {X 7.9802,Y -90.0317,Z 88,A -89.1608,B 24.9305,C -1.9247,E1 25.0154,E2 534.2417} C_DIS
LIN {X 9.9625,Y -89.8351,Z 88,A -87.8815,B 24.9305,C -1.926,E1 25.0189,E2 532.9602} C_DIS
LIN {X 12.5703,Y -89.5058,Z 88,A -86.0952,B 24.9301,C -1.9312,E1 25.0239,E2 531.1631} C_DIS
LIN {X 15.6753,Y -89.015,Z 88,A -84.2283,B 24.9303,C -1.9284,E1 25.029,E2 529.3047} C_DIS
LIN {X 18.2654,Y -88.5193,Z 88,A -82.4794,B 24.93,C -1.9325,E1 25.0338,E2 527.5482} C_DIS
LIN {X 20.8844,Y -87.9399,Z 88,A -80.8625,B 24.93,C -1.9312,E1 25.0382,E2 525.9367} C_DIS
LIN {X 23.2547,Y -87.3419,Z 88,A -79.4491,B 24.9303,C -1.9281,E1 25.042,E2 524.5327} C_DIS
LIN {X 25.3912,Y -86.7449,Z 88,A -78.0466,B 24.9303,C -1.9295,E1 25.0458,E2 523.1292} C_DIS
LIN {X 27.5124,Y -86.0956,Z 88,A -76.6435,B 24.9301,C -1.931,E1 25.0495,E2 521.725} C_DIS
LIN {X 29.7837,Y -85.336,Z 88,A -75.0753,B 24.9298,C -1.9347,E1 25.0537,E2 520.1513} C_DIS
LIN {X 31.9641,Y -84.5434,Z 88,A -73.4056,B 24.9292,C -1.9435,E1 25.0581,E2 518.4641} C_DIS
LIN {X 34.7977,Y -83.4177,Z 88,A -71.6037,B 24.9293,C -1.9417,E1 25.0627,E2 516.6706} C_DIS
LIN {X 37.8445,Y -82.0804,Z 88,A -69.3667,B 24.9288,C -1.9494,E1 25.0685,E2 514.421} C_DIS
LIN {X 40.6385,Y -80.7348,Z 88,A -67.4321,B 24.9286,C -1.9515,E1 25.0733,E2 512.4867} C_DIS
LIN {X 42.6076,Y -79.7131,Z 88,A -66.0312,B 24.9284,C -1.9537,E1 25.0768,E2 511.0846} C_DIS
LIN {X 45.5127,Y -78.0909,Z 88,A -63.9299,B 24.9282,C -1.9571,E1 25.0819,E2 508.9813} C_DIS
LIN {X 48.3562,Y -76.3628,Z 88,A -61.8294,B 24.9279,C -1.9608,E1 25.0869,E2 506.8787} C_DIS
LIN {X 50.403,Y -75.0261,Z 88,A -60.3963,B 24.9279,C -1.9597,E1 25.0902,E2 505.453} C_DIS
LIN {X 52.2291,Y -73.7666,Z 88,A -58.8893,B 24.9275,C -1.9662,E1 25.0937,E2 503.9359} C_DIS
LIN {X 54.7296,Y -71.9323,Z 88,A -57.0394,B 24.9275,C -1.9662,E1 25.0978,E2 502.0927} C_DIS
LIN {X 56.4784,Y -70.5675,Z 88,A -55.53,B 24.927,C -1.9729,E1 25.1011,E2 500.5731} C_DIS
LIN {X 58.6307,Y -68.7875,Z 88,A -53.7763,B 24.9268,C -1.9763,E1 25.1049,E2 498.8181} C_DIS
LIN {X 60.8661,Y -66.8184,Z 88,A -51.9992,B 24.9268,C -1.9766,E1 25.1085,E2 497.0473} C_DIS
LIN {X 63.2843,Y -64.5329,Z 88,A -50.0327,B 24.9268,C -1.9766,E1 25.1125,E2 495.0891} C_DIS
LIN {X 64.8489,Y -62.9603,Z 88,A -48.6341,B 24.9265,C -1.9797,E1 25.1153,E2 493.689} C_DIS
LIN {X 66.643,Y -61.0574,Z 88,A -46.7665,B 24.9256,C -1.9914,E1 25.1188,E2 491.802} C_DIS
LIN {X 68.7582,Y -58.6651,Z 88,A -44.71,B 24.9252,C -1.9977,E1 25.1226,E2 489.7398} C_DIS
LIN {X 70.7079,Y -56.3009,Z 88,A -43.0404,B 24.9255,C -1.993,E1 25.1255,E2 488.0891} C_DIS
LIN {X 71.9323,Y -54.7296,Z 88,A -41.5431,B 24.9246,C -2.0048,E1 25.1281,E2 486.571} C_DIS
LIN {X 73.2538,Y -52.9478,Z 88,A -40.2549,B 24.9246,C -2.0044,E1 25.1302,E2 485.29} C_DIS
LIN {X 74.5312,Y -51.1341,Z 88,A -38.8572,B 24.9244,C -2.0079,E1 25.1325,E2 483.8908} C_DIS
LIN {X 75.8858,Y -49.0992,Z 88,A -37.4492,B 24.9244,C -2.0072,E1 25.1346,E2 482.4916} C_DIS
LIN {X 77.1424,Y -47.0996,Z 88,A -35.8932,B 24.924,C -2.0135,E1 25.1369,E2 480.9285} C_DIS
LIN {X 78.6435,Y -44.551,Z 88,A -33.8564,B 24.9231,C -2.0248,E1 25.1398,E2 478.8755} C_DIS
LIN {X 79.7131,Y -42.6076,Z 88,A -32.459,B 24.9228,C -2.0286,E1 25.1416,E2 477.4765} C_DIS
LIN {X 80.7348,Y -40.6385,Z 88,A -31.0617,B 24.9225,C -2.0324,E1 25.1434,E2 476.0777} C_DIS
LIN {X 81.7078,Y -38.6449,Z 88,A -29.6648,B 24.9222,C -2.0363,E1 25.1451,E2 474.6791} C_DIS
LIN {X 82.6316,Y -36.6281,Z 88,A -28.2296,B 24.9218,C -2.0416,E1 25.1467,E2 473.2392} C_DIS
LIN {X 83.5909,Y -34.3795,Z 88,A -26.8381,B 24.9219,C -2.0406,E1 25.1482,E2 471.8579} C_DIS
LIN {X 84.7221,Y -31.4921,Z 88,A -24.7753,B 24.9212,C -2.0501,E1 25.1503,E2 469.784} C_DIS
LIN {X 85.8238,Y -28.3524,Z 88,A -22.6805,B 24.9207,C -2.0561,E1 25.1522,E2 467.6868} C_DIS
LIN {X 86.4938,Y -26.2376,Z 88,A -21.2836,B 24.9204,C -2.0602,E1 25.1533,E2 466.2883} C_DIS
LIN {X 87.2333,Y -23.6569,Z 88,A -19.566,B 24.9199,C -2.0661,E1 25.1546,E2 464.5664} C_DIS
LIN {X 87.9909,Y -20.6639,Z 88,A -17.7089,B 24.9198,C -2.0687,E1 25.1558,E2 462.7142} C_DIS
LIN {X 88.649,Y -17.6334,Z 88,A -15.6214,B 24.9189,C -2.0794,E1 25.157,E2 460.6135} C_DIS
LIN {X 89.0924,Y -15.2293,Z 88,A -14.2688,B 24.9191,C -2.0771,E1 25.1577,E2 459.2742} C_DIS
LIN {X 89.4223,Y -13.1579,Z 88,A -12.8907,B 24.9186,C -2.0831,E1 25.1583,E2 457.89} C_DIS
LIN {X 89.7324,Y -10.8394,Z 88,A -11.4757,B 24.9184,C -2.0854,E1 25.1588,E2 456.478} C_DIS
LIN {X 90.0705,Y -7.5293,Z 88,A -9.5135,B 24.9184,C -2.0868,E1 25.1593,E2 454.5241} C_DIS
LIN {X 90.2282,Y -5.3166,Z 88,A -8.1171,B 24.918,C -2.091,E1 25.1595,E2 453.1262} C_DIS
LIN {X 90.3315,Y -3.1006,Z 88,A -6.7208,B 24.9177,C -2.0951,E1 25.1597,E2 451.7284} C_DIS
LIN {X 90.379,Y -1.1092,Z 88,A -5.0966,B 24.9163,C -2.1123,E1 25.1597,E2 450.0732} C_DIS
LIN {X 90.3586,Y 2.2182,Z 88,A -3.2398,B 24.9165,C -2.1099,E1 25.1597,E2 448.2332} C_DIS
LIN {X 90.2769,Y 4.435,Z 88,A -1.7336,B 24.9159,C -2.118,E1 25.1595,E2 446.7168} C_DIS
LIN {X 90.1409,Y 6.6492,Z 88,A -0.3369,B 24.9155,C -2.1221,E1 25.1592,E2 445.3187} C_DIS
LIN {X 89.9506,Y 8.8594,Z 88,A 0.9499,B 24.9155,C -2.1222,E1 25.1589,E2 444.0393} C_DIS
LIN {X 89.677,Y 11.2886,Z 88,A 2.4886,B 24.9152,C -2.1267,E1 25.1584,E2 442.4991} C_DIS
LIN {X 89.238,Y 14.3585,Z 88,A 4.672,B 24.914,C -2.1408,E1 25.1575,E2 440.2953} C_DIS
LIN {X 88.649,Y 17.6334,Z 88,A 6.7338,B 24.9137,C -2.1456,E1 25.1564,E2 438.2341} C_DIS
LIN {X 87.9399,Y 20.8844,Z 88,A 8.7411,B 24.9134,C -2.1484,E1 25.1552,E2 436.2319} C_DIS
LIN {X 87.3889,Y 23.0807,Z 88,A 10.144,B 24.9132,C -2.1516,E1 25.1542,E2 434.8296} C_DIS
LIN {X 86.4938,Y 26.2376,Z 88,A 12.2336,B 24.9126,C -2.1582,E1 25.1525,E2 432.7363} C_DIS
LIN {X 85.8239,Y 28.3524,Z 88,A 13.5209,B 24.9126,C -2.1581,E1 25.1514,E2 431.4565} C_DIS
LIN {X 84.8892,Y 31.034,Z 88,A 15.3963,B 24.912,C -2.1661,E1 25.1497,E2 429.5727} C_DIS
LIN {X 83.8384,Y 33.7714,Z 88,A 17.1565,B 24.9118,C -2.168,E1 25.1479,E2 427.8179} C_DIS
LIN {X 82.6316,Y 36.6281,Z 88,A 19.2201,B 24.9111,C -2.1771,E1 25.1456,E2 425.7441} C_DIS
LIN {X 81.5302,Y 39.0144,Z 88,A 20.8982,B 24.9107,C -2.1822,E1 25.1436,E2 424.0629} C_DIS
LIN {X 80.1245,Y 41.8264,Z 88,A 22.7468,B 24.9107,C -2.1825,E1 25.1412,E2 422.2234} C_DIS
LIN {X 78.5307,Y 44.7472,Z 88,A 24.9974,B 24.9098,C -2.1933,E1 25.1382,E2 419.9592} C_DIS
LIN {X 76.8305,Y 47.6074,Z 88,A 26.8086,B 24.9102,C -2.1882,E1 25.1356,E2 418.1692} C_DIS
LIN {X 75.7636,Y 49.2896,Z 88,A 28.3066,B 24.9092,C -2.1998,E1 25.1333,E2 416.6513} C_DIS
LIN {X 73.898,Y 52.0449,Z 88,A 30.4043,B 24.9088,C -2.2047,E1 25.13,E2 414.5523} C_DIS
LIN {X 71.9323,Y 54.7296,Z 88,A 32.5024,B 24.9084,C -2.2095,E1 25.1265,E2 412.453} C_DIS
LIN {X 70.4251,Y 56.6542,Z 88,A 34.0652,B 24.9081,C -2.2136,E1 25.1237,E2 410.8877} C_DIS
LIN {X 68.4409,Y 59.0375,Z 88,A 36,B 24.9078,C -2.2171,E1 25.1202,E2 408.9537} C_DIS
LIN {X 66.9715,Y 60.6994,Z 88,A 37.2893,B 24.9078,C -2.2161,E1 25.1179,E2 407.6723} C_DIS
LIN {X 65.4616,Y 62.3247,Z 88,A 38.7987,B 24.9073,C -2.2228,E1 25.1149,E2 406.1536} C_DIS
LIN {X 63.9124,Y 63.9124,Z 88,A 40.1984,B 24.9071,C -2.2256,E1 25.1122,E2 404.7533} C_DIS
LIN {X 62.3247,Y 65.4616,Z 88,A 41.4885,B 24.9071,C -2.2244,E1 25.1096,E2 403.4714} C_DIS
LIN {X 60.6994,Y 66.9714,Z 88,A 43.1172,B 24.9063,C -2.235,E1 25.1062,E2 401.8241} C_DIS
LIN {X 58.1932,Y 69.1602,Z 88,A 45.0987,B 24.9063,C -2.2346,E1 25.102,E2 399.8513} C_DIS
LIN {X 56.4784,Y 70.5675,Z 88,A 46.3893,B 24.9064,C -2.2332,E1 25.0992,E2 398.569} C_DIS
LIN {X 54.7296,Y 71.9323,Z 88,A 47.79,B 24.9062,C -2.2355,E1 25.0961,E2 397.1679} C_DIS
LIN {X 52.9478,Y 73.2538,Z 88,A 49.191,B 24.9061,C -2.2378,E1 25.093,E2 395.7665} C_DIS
LIN {X 50.9467,Y 74.658,Z 88,A 50.7349,B 24.9059,C -2.2402,E1 25.0894,E2 394.2223} C_DIS
LIN {X 48.3562,Y 76.3628,Z 88,A 52.6943,B 24.9056,C -2.243,E1 25.0848,E2 392.2625} C_DIS
LIN {X 46.4676,Y 77.5265,Z 88,A 54.0957,B 24.9055,C -2.2449,E1 25.0815,E2 390.861} C_DIS
LIN {X 44.2921,Y 78.7881,Z 88,A 55.7204,B 24.9052,C -2.2483,E1 25.0776,E2 389.2332} C_DIS
LIN {X 41.8264,Y 80.1245,Z 88,A 57.48,B 24.905,C -2.25,E1 25.0732,E2 387.4745} C_DIS
LIN {X 39.4407,Y 81.3254,Z 88,A 59.0135,B 24.9053,C -2.2467,E1 25.0694,E2 385.953} C_DIS
LIN {X 37.4001,Y 82.2836,Z 88,A 60.4176,B 24.9053,C -2.2475,E1 25.0659,E2 384.5505} C_DIS
LIN {X 35.6113,Y 83.0748,Z 88,A 61.9191,B 24.9044,C -2.2577,E1 25.062,E2 383.0285} C_DIS
LIN {X 33.5618,Y 83.9238,Z 88,A 63.3223,B 24.9043,C -2.259,E1 25.0583,E2 381.6253} C_DIS
LIN {X 31.4921,Y 84.7221,Z 88,A 64.7255,B 24.9042,C -2.2603,E1 25.0547,E2 380.2223} C_DIS
LIN {X 29.189,Y 85.5418,Z 88,A 66.1618,B 24.9044,C -2.2578,E1 25.0509,E2 378.7947} C_DIS
LIN {X 26.2376,Y 86.4938,Z 88,A 68.2348,B 24.9039,C -2.2629,E1 25.0454,E2 376.7133} C_DIS
LIN {X 24.107,Y 87.1117,Z 88,A 69.5287,B 24.9042,C -2.2601,E1 25.0419,E2 375.4282} C_DIS
LIN {X 21.7421,Y 87.7307,Z 88,A 71.0763,B 24.9041,C -2.261,E1 25.0377,E2 373.8809} C_DIS
LIN {X 18.7199,Y 88.426,Z 88,A 73.1504,B 24.9037,C -2.2655,E1 25.032,E2 371.7987} C_DIS
LIN {X 16.5442,Y 88.8588,Z 88,A 74.5555,B 24.9037,C -2.2661,E1 25.0282,E2 370.3939} C_DIS
LIN {X 13.2623,Y 89.4075,Z 88,A 76.7069,B 24.9035,C -2.2681,E1 25.0222,E2 368.2398} C_DIS
LIN {X 10.8394,Y 89.7324,Z 88,A 78.1019,B 24.9039,C -2.2633,E1 25.0184,E2 366.8573} C_DIS
LIN {X 7.5293,Y 90.0705,Z 88,A 80.0773,B 24.9043,C -2.2592,E1 25.013,E2 364.893} C_DIS
LIN {X 5.3166,Y 90.2282,Z 88,A 81.4835,B 24.9043,C -2.2592,E1 25.009,E2 363.4873} C_DIS
LIN {X 3.1006,Y 90.3315,Z 88,A 83.1595,B 24.9035,C -2.2679,E1 25.0043,E2 361.791} C_DIS
LIN {X 0,Y 90.3858,Z 88,A 85.1004,B 24.9036,C -2.2668,E1 24.9989,E2 359.8531} C_DIS
LIN {X -2.2182,Y 90.3586,Z 88,A 86.5079,B 24.9036,C -2.2664,E1 24.995,E2 358.4462} C_DIS
LIN {X -4.435,Y 90.2769,Z 88,A 87.915,B 24.9036,C -2.266,E1 24.991,E2 357.0399} C_DIS
LIN {X -6.6492,Y 90.1409,Z 88,A 89.3228,B 24.9037,C -2.2655,E1 24.9871,E2 355.6329} C_DIS
LIN {X -8.8594,Y 89.9506,Z 88,A 90.6198,B 24.9041,C -2.2612,E1 24.9835,E2 354.3451} C_DIS
LIN {X -11.2886,Y 89.677,Z 88,A 92.1711,B 24.9041,C -2.2604,E1 24.9792,E2 352.7947} C_DIS
LIN {X -14.6094,Y 89.1961,Z 88,A 94.2887,B 24.9043,C -2.2587,E1 24.9734,E2 350.6795} C_DIS
LIN {X -16.7664,Y 88.816,Z 88,A 95.6925,B 24.9043,C -2.2581,E1 24.9695,E2 349.2756} C_DIS
LIN {X -19.8036,Y 88.1896,Z 88,A 97.6621,B 24.9045,C -2.2565,E1 24.9642,E2 347.3073} C_DIS
LIN {X -21.962,Y 87.677,Z 88,A 99.2846,B 24.904,C -2.2621,E1 24.9597,E2 345.6694} C_DIS
LIN {X -25.1742,Y 86.8093,Z 88,A 101.1852,B 24.9048,C -2.2533,E1 24.9547,E2 343.7868} C_DIS
LIN {X -27.5124,Y 86.0956,Z 88,A 102.6055,B 24.9052,C -2.2474,E1 24.9509,E2 342.3778} C_DIS
LIN {X -29.4034,Y 85.4695,Z 88,A 104.116,B 24.9047,C -2.2537,E1 24.9469,E2 340.8496} C_DIS
LIN {X -31.4921,Y 84.7221,Z 88,A 105.4155,B 24.9052,C -2.2485,E1 24.9435,E2 339.5598} C_DIS
LIN {X -33.5618,Y 83.9238,Z 88,A 106.9369,B 24.905,C -2.2502,E1 24.9395,E2 338.031} C_DIS
LIN {X -36.6281,Y 82.6316,Z 88,A 109.0531,B 24.9052,C -2.2474,E1 24.9341,E2 335.9166} C_DIS
LIN {X -38.6449,Y 81.7078,Z 88,A 110.4639,B 24.9054,C -2.2454,E1 24.9305,E2 334.507} C_DIS
LIN {X -40.84,Y 80.6318,Z 88,A 111.9082,B 24.9059,C -2.2397,E1 24.9269,E2 333.0726} C_DIS
LIN {X -43.1658,Y 79.4103,Z 88,A 113.6634,B 24.9059,C -2.2397,E1 24.9226,E2 331.3124} C_DIS
LIN {X -45.7075,Y 77.9757,Z 88,A 115.3035,B 24.9067,C -2.2299,E1 24.9187,E2 329.6908} C_DIS
LIN {X -47.6074,Y 76.8305,Z 88,A 116.7153,B 24.9069,C -2.2275,E1 24.9153,E2 328.2803} C_DIS
LIN {X -49.7954,Y 75.4301,Z 88,A 118.5956,B 24.9066,C -2.2316,E1 24.9109,E2 326.3842} C_DIS
LIN {X -52.4349,Y 73.6198,Z 88,A 120.6756,B 24.9068,C -2.2291,E1 24.9061,E2 324.303} C_DIS
LIN {X -54.9089,Y 71.7942,Z 88,A 122.3649,B 24.9078,C -2.2171,E1 24.9024,E2 322.6363} C_DIS
LIN {X -56.4784,Y 70.5675,Z 88,A 123.7675,B 24.9077,C -2.2186,E1 24.8993,E2 321.2248} C_DIS
LIN {X -58.1932,Y 69.1602,Z 88,A 125.2919,B 24.9077,C -2.2192,E1 24.896,E2 319.6933} C_DIS
LIN {X -60.0416,Y 67.5603,Z 88,A 126.7695,B 24.9081,C -2.2135,E1 24.8929,E2 318.2234} C_DIS
LIN {X -61.6815,Y 66.0665,Z 88,A 128.1516,B 24.9084,C -2.2095,E1 24.8901,E2 316.8452} C_DIS
LIN {X -63.9124,Y 63.9124,Z 88,A 130.2644,B 24.9084,C -2.2093,E1 24.8859,E2 314.7241} C_DIS
LIN {X -65.6167,Y 62.1598,Z 88,A 131.6861,B 24.9091,C -2.2016,E1 24.8831,E2 313.3145} C_DIS
LIN {X -67.1224,Y 60.5308,Z 88,A 133.0999,B 24.9093,C -2.1983,E1 24.8805,E2 311.9022} C_DIS
LIN {X -68.5076,Y 58.9593,Z 88,A 134.3747,B 24.9098,C -2.1934,E1 24.8782,E2 310.6335} C_DIS
LIN {X -69.8692,Y 57.3401,Z 88,A 135.7843,B 24.9098,C -2.1919,E1 24.8756,E2 309.2208} C_DIS
LIN {X -71.3934,Y 55.4289,Z 88,A 137.2088,B 24.9105,C -2.1841,E1 24.8732,E2 307.8083} C_DIS
LIN {X -72.7093,Y 53.6915,Z 88,A 138.7512,B 24.9105,C -2.1852,E1 24.8706,E2 306.2558} C_DIS
LIN {X -74.5312,Y 51.1341,Z 88,A 140.7352,B 24.9109,C -2.1796,E1 24.8674,E2 304.2754} C_DIS
LIN {X -75.7636,Y 49.2896,Z 88,A 142.1616,B 24.9112,C -2.1763,E1 24.8652,E2 302.8498} C_DIS
LIN {X -76.9504,Y 47.4154,Z 88,A 143.6765,B 24.9112,C -2.1756,E1 24.863,E2 301.3288} C_DIS
LIN {X -78.0909,Y 45.5127,Z 88,A 145.0918,B 24.9115,C -2.1718,E1 24.861,E2 299.9152} C_DIS
LIN {X -79.1843,Y 43.5826,Z 88,A 146.3956,B 24.9121,C -2.1647,E1 24.8592,E2 298.6215} C_DIS
LIN {X -80.463,Y 41.1703,Z 88,A 148.2612,B 24.9121,C -2.1637,E1 24.8568,E2 296.7484} C_DIS
LIN {X -81.7078,Y 38.6449,Z 88,A 150.0456,B 24.9126,C -2.1584,E1 24.8546,E2 294.9671} C_DIS
LIN {X -82.6316,Y 36.6281,Z 88,A 151.3499,B 24.9132,C -2.1511,E1 24.8532,E2 293.6729} C_DIS
LIN {X -83.5056,Y 34.5891,Z 88,A 152.7655,B 24.9135,C -2.1471,E1 24.8516,E2 292.2589} C_DIS
LIN {X -84.3293,Y 32.5294,Z 88,A 154.2925,B 24.9135,C -2.1465,E1 24.8501,E2 290.725} C_DIS
LIN {X -85.1022,Y 30.4501,Z 88,A 155.7086,B 24.9139,C -2.1424,E1 24.8487,E2 289.3106} C_DIS
LIN {X -85.8238,Y 28.3524,Z 88,A 157.1243,B 24.9142,C -2.1384,E1 24.8475,E2 287.8964} C_DIS
LIN {X -86.4938,Y 26.2376,Z 88,A 158.6205,B 24.9144,C -2.1366,E1 24.8463,E2 286.3958} C_DIS
LIN {X -87.2276,Y 23.6777,Z 88,A 160.2402,B 24.915,C -2.1293,E1 24.845,E2 284.784} C_DIS
LIN {X -87.9909,Y 20.6639,Z 88,A 161.9792,B 24.916,C -2.1163,E1 24.8439,E2 283.0661} C_DIS
LIN {X -88.4715,Y 18.4982,Z 88,A 163.5295,B 24.916,C -2.1161,E1 24.843,E2 281.5072} C_DIS
LIN {X -89.0924,Y 15.2293,Z 88,A 165.6536,B 24.9165,C -2.1098,E1 24.8419,E2 279.3854} C_DIS
LIN {X -89.6298,Y 11.6524,Z 88,A 168.0854,B 24.9168,C -2.1066,E1 24.841,E2 276.9467} C_DIS
LIN {X -89.9506,Y 8.8594,Z 88,A 169.8696,B 24.9172,C -2.1009,E1 24.8404,E2 275.1654} C_DIS
LIN {X -90.1409,Y 6.6492,Z 88,A 171.286,B 24.9176,C -2.0967,E1 24.8401,E2 273.7506} C_DIS
LIN {X -90.3245,Y 3.3268,Z 88,A 173.2986,B 24.9183,C -2.0871,E1 24.8399,E2 271.7487} C_DIS
LIN {X -90.3819,Y 0.7187,Z 88,A 175.1483,B 24.9183,C -2.0876,E1 24.8398,E2 269.8866} C_DIS
LIN {X -90.3586,Y -2.2182,Z 88,A 176.9507,B 24.9189,C -2.0799,E1 24.8398,E2 268.0918} C_DIS
LIN {X -90.2769,Y -4.435,Z 88,A 178.3667,B 24.9192,C -2.0757,E1 24.8401,E2 266.6773} C_DIS
LIN {X -90.0932,Y -7.2451,Z 88,A -179.8515,B 24.9196,C -2.07,E1 24.8404,E2 264.8985} C_DIS
LIN {X -89.8351,Y -9.9625,Z 88,A -178.2043,B 24.9203,C -2.062,E1 24.8409,E2 263.2605} C_DIS
LIN {X -89.5317,Y -12.3882,Z 88,A -176.778,B 24.9209,C -2.0535,E1 24.8414,E2 261.8459} C_DIS
LIN {X -89.2284,Y -14.4162,Z 88,A -175.253,B 24.9207,C -2.0561,E1 24.8421,E2 260.3056} C_DIS
LIN {X -88.816,Y -16.7664,Z 88,A -173.8119,B 24.9212,C -2.0493,E1 24.8428,E2 258.8722} C_DIS
LIN {X -88.3099,Y -19.252,Z 88,A -172.0804,B 24.9213,C -2.0481,E1 24.8438,E2 257.1335} C_DIS
LIN {X -87.677,Y -21.962,Z 88,A -170.3056,B 24.9217,C -2.043,E1 24.8449,E2 255.3604} C_DIS
LIN {X -87.1117,Y -24.107,Z 88,A -168.8898,B 24.922,C -2.039,E1 24.846,E2 253.9459} C_DIS
LIN {X -86.4938,Y -26.2376,Z 88,A -167.4741,B 24.9223,C -2.0351,E1 24.8471,E2 252.5315} C_DIS
LIN {X -85.8045,Y -28.4098,Z 88,A -166.1671,B 24.923,C -2.0266,E1 24.8482,E2 251.2371} C_DIS
LIN {X -84.9746,Y -30.7998,Z 88,A -164.3796,B 24.923,C -2.0275,E1 24.8499,E2 249.4375} C_DIS
LIN {X -83.9238,Y -33.5618,Z 88,A -162.5203,B 24.9234,C -2.0216,E1 24.8518,E2 247.5818} C_DIS
LIN {X -82.7829,Y -36.2808,Z 88,A -160.5848,B 24.9236,C -2.0183,E1 24.8539,E2 245.6434} C_DIS
LIN {X -81.5618,Y -38.9487,Z 88,A -158.9297,B 24.9245,C -2.0069,E1 24.8559,E2 244.0066} C_DIS
LIN {X -80.1245,Y -41.8264,Z 88,A -156.9613,B 24.9251,C -1.9991,E1 24.8583,E2 242.0461} C_DIS
LIN {X -79.0739,Y -43.7801,Z 88,A -155.3218,B 24.9248,C -2.0024,E1 24.8606,E2 240.3901} C_DIS
LIN {X -77.6416,Y -46.2728,Z 88,A -153.4459,B 24.9251,C -1.9992,E1 24.8632,E2 238.5121} C_DIS
LIN {X -76.3628,Y -48.3562,Z 88,A -151.9099,B 24.9254,C -1.9947,E1 24.8655,E2 236.9789} C_DIS
LIN {X -75.0261,Y -50.403,Z 88,A -150.4627,B 24.9259,C -1.9877,E1 24.8677,E2 235.5413} C_DIS
LIN {X -73.7666,Y -52.2291,Z 88,A -149.0721,B 24.9262,C -1.9837,E1 24.8699,E2 234.1534} C_DIS
LIN {X -72.2239,Y -54.3415,Z 88,A -147.2942,B 24.9262,C -1.9833,E1 24.8729,E2 232.3677} C_DIS
LIN {X -70.4279,Y -56.6507,Z 88,A -145.5151,B 24.9267,C -1.9766,E1 24.876,E2 230.5962} C_DIS
LIN {X -68.4409,Y -59.0375,Z 88,A -143.3098,B 24.9265,C -1.9794,E1 24.88,E2 228.3744} C_DIS
LIN {X -66.2215,Y -61.5167,Z 88,A -141.3203,B 24.9272,C -1.971,E1 24.8837,E2 226.396} C_DIS
LIN {X -63.9124,Y -63.9124,Z 88,A -139.1883,B 24.9274,C -1.9672,E1 24.8879,E2 224.2639} C_DIS
LIN {X -62.3247,Y -65.4616,Z 88,A -137.8865,B 24.9279,C -1.9611,E1 24.8905,E2 222.9713} C_DIS
LIN {X -60.5308,Y -67.1224,Z 88,A -136.3304,B 24.9281,C -1.9582,E1 24.8937,E2 221.4157} C_DIS
LIN {X -58.8653,Y -68.5877,Z 88,A -134.8804,B 24.9282,C -1.9569,E1 24.8967,E2 219.9633} C_DIS
LIN {X -57.1643,Y -70.0116,Z 88,A -133.3741,B 24.9282,C -1.9574,E1 24.9,E2 218.45} C_DIS
LIN {X -54.7296,Y -71.9323,Z 88,A -131.4213,B 24.9285,C -1.9535,E1 24.9043,E2 216.4994} C_DIS
LIN {X -52.9478,Y -73.2538,Z 88,A -130.1205,B 24.9289,C -1.9477,E1 24.9072,E2 215.2077} C_DIS
LIN {X -51.1341,Y -74.5312,Z 88,A -128.7093,B 24.929,C -1.9456,E1 24.9105,E2 213.7968} C_DIS
LIN {X -49.0992,Y -75.8858,Z 88,A -127.2877,B 24.9295,C -1.9391,E1 24.9137,E2 212.3859} C_DIS
LIN {X -47.0361,Y -77.1809,Z 88,A -125.7007,B 24.9295,C -1.9382,E1 24.9175,E2 210.7962} C_DIS
LIN {X -44.551,Y -78.6435,Z 88,A -123.6607,B 24.9293,C -1.9423,E1 24.9225,E2 208.7402} C_DIS
LIN {X -42.6076,Y -79.7131,Z 88,A -122.2502,B 24.9293,C -1.9406,E1 24.9259,E2 207.3298} C_DIS
LIN {X -40.1095,Y -80.997,Z 88,A -120.4783,B 24.9296,C -1.9382,E1 24.9304,E2 205.559} C_DIS
LIN {X -37.433,Y -82.2688,Z 88,A -118.8258,B 24.9303,C -1.9287,E1 24.9345,E2 203.9248} C_DIS
LIN {X -35.0698,Y -83.303,Z 88,A -116.955,B 24.9298,C -1.9346,E1 24.9393,E2 202.0357} C_DIS
LIN {X -32.3178,Y -84.4094,Z 88,A -115.3025,B 24.9305,C -1.9254,E1 24.9436,E2 200.4013} C_DIS
LIN {X -30.2365,Y -85.1771,Z 88,A -113.7601,B 24.9303,C -1.9286,E1 24.9477,E2 198.8483} C_DIS
LIN {X -27.0809,Y -86.2323,Z 88,A -111.7805,B 24.9307,C -1.9228,E1 24.9529,E2 196.879} C_DIS
LIN {X -24.9565,Y -86.871,Z 88,A -110.3719,B 24.9307,C -1.9219,E1 24.9567,E2 195.4702} C_DIS
LIN {X -22.817,Y -87.4573,Z 88,A -108.8306,B 24.9305,C -1.9254,E1 24.9608,E2 193.918} C_DIS
LIN {X -20.51,Y -88.0264,Z 88,A -107.19,B 24.9302,C -1.929,E1 24.9653,E2 192.2666} C_DIS
Enddeposition()
END
